// TIA Portal project "Control and SCADA Codes" (V20)
// Source code materials for the Control and SCADA Systems course.

(* hardware
DEVICE "S7-1500/ET200MP station_1"  S7-1500 station
   slot 0: "Rail_0"  Rack  6ES7 590-1***0-0AA0
   slot 1: "Control"  CPU 1511-1 PN  6ES7 511-1AL03-0AB0  V4.0
      slot 3: "CPU display_1"  6ES7591-1AA00-0AA0
      slot 32768: "PROFINET interface_1"  X1
         slot 32769: "Port_1"  X1 P1
         slot 32770: "Port_2"  X1 P2
      slot 34817: "Virtual CP interface port_1"  Virtual CP interface port  Virtual CP interface port FW V4.0
DEVICE "SCADA"  SIMATIC PC station
   slot 0: "SIMATIC PC station"  Rail  SIMATIC PC-Station  V1.0
      slot 125: "Stationmanager"  Station_Manager  V6.0.4
   slot 1: "HMI_RT_1"  WinCC Unified PC RT  6AV2 155-xxxxx-xxxx  20.0.0.0
DEVICE "S7-1500/ET200MP station_2"  S7-1500 station
   slot 0: "Rail_0"  Rack  6ES7 590-1***0-0AA0
   slot 1: "State Diagram Controller"  CPU 1511-1 PN  6ES7 511-1AL03-0AB0  V4.0
      slot 3: "CPU display_1"  6ES7591-1AA00-0AA0
      slot 32768: "PROFINET interface_1"  X1
         slot 32769: "Port_1"  X1 P1
         slot 32770: "Port_2"  X1 P2
      slot 34817: "Virtual CP interface port_1"  Virtual CP interface port  Virtual CP interface port FW V4.0
DEVICE "State Diagram SCADA"  SIMATIC PC station
   slot 0: "SIMATIC PC station"  Rail  SIMATIC PC-Station  V1.0
      slot 125: "Stationmanager"  Station_Manager  V6.0.4
   slot 1: "HMI_RT_2"  WinCC Unified PC RT  6AV2 155-xxxxx-xxxx  20.0.0.0
DEVICE "S7-1500/ET200MP station_3"  S7-1500 station
   slot 0: "Rail_0"  Rack  6ES7 590-1***0-0AA0
   slot 1: "OOP Controller"  CPU 1511-1 PN  6ES7 511-1AL03-0AB0  V4.0
      slot 3: "CPU display_1"  6ES7591-1AA00-0AA0
      slot 32768: "PROFINET interface_1"  X1
         slot 32769: "Port_1"  X1 P1
         slot 32770: "Port_2"  X1 P2
      slot 34817: "Virtual CP interface port_1"  Virtual CP interface port  Virtual CP interface port FW V4.0
DEVICE "OOP SCADA"  SIMATIC PC station
   slot 0: "SIMATIC PC station"  Rail  SIMATIC PC-Station  V1.0
      slot 125: "Stationmanager"  Station_Manager  V6.0.4
   slot 1: "HMI_RT_3"  WinCC Unified PC RT  6AV2 155-xxxxx-xxxx  20.0.0.0
DEVICE "S7-1500/ET200MP station_4"  S7-1500 station
   slot 0: "Rail_0"  Rack  6ES7 590-1***0-0AA0
   slot 1: "Contiuous Controller"  CPU 1511-1 PN  6ES7 511-1AL03-0AB0  V4.0
      slot 3: "CPU display_1"  6ES7591-1AA00-0AA0
      slot 32768: "PROFINET interface_1"  X1
         slot 32769: "Port_1"  X1 P1
         slot 32770: "Port_2"  X1 P2
      slot 34817: "Virtual CP interface port_1"  Virtual CP interface port  Virtual CP interface port FW V4.0
DEVICE "Continuous Ctrl SCADA"  SIMATIC PC station
   slot 0: "SIMATIC PC station"  Rail  SIMATIC PC-Station  V1.0
      slot 125: "Stationmanager"  Station_Manager  V6.0.4
   slot 1: "HMI_RT_4"  WinCC Unified PC RT  6AV2 155-xxxxx-xxxx  20.0.0.0
DEVICE "PC-System_1"  SIMATIC PC station
   slot 0: "SIMATIC PC station"  Rail  SIMATIC PC-Station  V1.0
      slot 125: "Stationmanager"  Station_Manager  V6.0.4
   slot 1: "Energy Management"  WinCC Unified PC RT  6AV2 155-xxxxx-xxxx  20.0.0.0
*)

// ===== PLC "Control"  CPU 1511-1 PN =====

VAR_GLOBAL   // PLC tag table "01.MotorCtrl"
   "Start" AT %M0.0 : Bool;
   "Stop" AT %M0.1 : Bool;
   "Motor" AT %M0.2 : Bool;
   "Clock_Byte" AT %MB100 : Byte;
   "Clock_10Hz" AT %M100.0 : Bool;
   "Clock_5Hz" AT %M100.1 : Bool;
   "Clock_2.5Hz" AT %M100.2 : Bool;
   "Clock_2Hz" AT %M100.3 : Bool;
   "Clock_1.25Hz" AT %M100.4 : Bool;
   "Clock_1Hz" AT %M100.5 : Bool;
   "Clock_0.625Hz" AT %M100.6 : Bool;
   "Clock_0.5Hz" AT %M100.7 : Bool;
END_VAR

VAR_GLOBAL   // PLC tag table "02.ThreeSwitchesCtrlPump"
   "K1" AT %M0.3 : Bool;
   "K2" AT %M0.4 : Bool;
   "K3" AT %M0.5 : Bool;
   "Pump" AT %M0.6 : Bool;
END_VAR

VAR_GLOBAL CONSTANT   // PLC tag table "02.ThreeSwitchesCtrlPump"
   "None(1)" : Pip := 65535;
   "Automatic update(1)" : Pip := 0;
   "PIP 1(1)" : Pip := 1;
   "PIP 2(1)" : Pip := 2;
   "PIP 3(1)" : Pip := 3;
   "PIP 4(1)" : Pip := 4;
   "PIP 5(1)" : Pip := 5;
   "PIP 6(1)" : Pip := 6;
   "PIP 7(1)" : Pip := 7;
   "PIP 8(1)" : Pip := 8;
   "PIP 9(1)" : Pip := 9;
   "PIP 10(1)" : Pip := 10;
   "PIP 11(1)" : Pip := 11;
   "PIP 12(1)" : Pip := 12;
   "PIP 13(1)" : Pip := 13;
   "PIP 14(1)" : Pip := 14;
   "PIP 15(1)" : Pip := 15;
   "PIP 16(1)" : Pip := 16;
   "PIP 17(1)" : Pip := 17;
   "PIP 18(1)" : Pip := 18;
   "PIP 19(1)" : Pip := 19;
   "PIP 20(1)" : Pip := 20;
   "PIP 21(1)" : Pip := 21;
   "PIP 22(1)" : Pip := 22;
   "PIP 23(1)" : Pip := 23;
   "PIP 24(1)" : Pip := 24;
   "PIP 25(1)" : Pip := 25;
   "PIP 26(1)" : Pip := 26;
   "PIP 27(1)" : Pip := 27;
   "PIP 28(1)" : Pip := 28;
   "PIP 29(1)" : Pip := 29;
   "PIP 30(1)" : Pip := 30;
   "PIP 31(1)" : Pip := 31;
   "PIP OB Servo(1)" : Pip := 32768;
   "Local~MC(1)" : Hw_SubModule := 51;
   "Local~Common(1)" : Hw_SubModule := 50;
   "Local~Device(1)" : Hw_Device := 32;
   "Local~Configuration(1)" : Hw_SubModule := 33;
   "Local~Display(1)" : Hw_SubModule := 54;
   "Local~Exec(1)" : Hw_SubModule := 52;
   "Local(1)" : Hw_SubModule := 49;
   "Local~PROFINET_interface_1(1)" : Hw_Interface := 64;
   "Local~PROFINET_interface_1~Port_1(1)" : Hw_Interface := 65;
   "Local~PROFINET_interface_1~Port_2(1)" : Hw_Interface := 66;
   "Local~Virtual_communication_interface(1)" : Hw_Interface := 135;
   "Local~License_Manager(1)" : Hw_SubModule := 42;
   "OB_01. MotorCtrl_LD(1)" : OB_PCYCLE := 1;
   "OB_02. MotorCtrl_FBD(1)" : OB_PCYCLE := 124;
   "OB_03. MotorCtrl_ST(1)" : OB_PCYCLE := 123;
   "OB_01_TheeSwitchesCtrlPump_1(1)" : OB_PCYCLE := 125;
END_VAR

VAR_GLOBAL   // PLC tag table "03.SBO"
   "Select" AT %M0.7 : Bool;
   "Confirm" AT %M1.0 : Bool;
   "CB" AT %M1.1 : Bool;
END_VAR

VAR_GLOBAL CONSTANT   // PLC tag table "03.SBO"
   "None(2)" : Pip := 65535;
   "Automatic update(2)" : Pip := 0;
   "PIP 1(2)" : Pip := 1;
   "PIP 2(2)" : Pip := 2;
   "PIP 3(2)" : Pip := 3;
   "PIP 4(2)" : Pip := 4;
   "PIP 5(2)" : Pip := 5;
   "PIP 6(2)" : Pip := 6;
   "PIP 7(2)" : Pip := 7;
   "PIP 8(2)" : Pip := 8;
   "PIP 9(2)" : Pip := 9;
   "PIP 10(2)" : Pip := 10;
   "PIP 11(2)" : Pip := 11;
   "PIP 12(2)" : Pip := 12;
   "PIP 13(2)" : Pip := 13;
   "PIP 14(2)" : Pip := 14;
   "PIP 15(2)" : Pip := 15;
   "PIP 16(2)" : Pip := 16;
   "PIP 17(2)" : Pip := 17;
   "PIP 18(2)" : Pip := 18;
   "PIP 19(2)" : Pip := 19;
   "PIP 20(2)" : Pip := 20;
   "PIP 21(2)" : Pip := 21;
   "PIP 22(2)" : Pip := 22;
   "PIP 23(2)" : Pip := 23;
   "PIP 24(2)" : Pip := 24;
   "PIP 25(2)" : Pip := 25;
   "PIP 26(2)" : Pip := 26;
   "PIP 27(2)" : Pip := 27;
   "PIP 28(2)" : Pip := 28;
   "PIP 29(2)" : Pip := 29;
   "PIP 30(2)" : Pip := 30;
   "PIP 31(2)" : Pip := 31;
   "PIP OB Servo(2)" : Pip := 32768;
   "Local~MC(2)" : Hw_SubModule := 51;
   "Local~Common(2)" : Hw_SubModule := 50;
   "Local~Device(2)" : Hw_Device := 32;
   "Local~Configuration(2)" : Hw_SubModule := 33;
   "Local~Display(2)" : Hw_SubModule := 54;
   "Local~Exec(2)" : Hw_SubModule := 52;
   "Local(2)" : Hw_SubModule := 49;
   "Local~PROFINET_interface_1(2)" : Hw_Interface := 64;
   "Local~PROFINET_interface_1~Port_1(2)" : Hw_Interface := 65;
   "Local~PROFINET_interface_1~Port_2(2)" : Hw_Interface := 66;
   "Local~Virtual_communication_interface(2)" : Hw_Interface := 135;
   "Local~License_Manager(2)" : Hw_SubModule := 42;
   "OB_01.MotorCtrl_LD(1)" : OB_PCYCLE := 1;
   "OB_02.MotorCtrl_FBD(1)" : OB_PCYCLE := 124;
   "OB_03.MotorCtrl_ST(1)" : OB_PCYCLE := 123;
   "OB_01_TheeSwitchesCtrlPump_1(2)" : OB_PCYCLE := 125;
   "OB_02_TheeSwitchesCtrlPump_2(1)" : OB_PCYCLE := 126;
   "OB_02.SBO_ST(1)" : OB_PCYCLE := 123;
   "OB_01.SBO_LD(1)" : OB_PCYCLE := 1;
END_VAR

VAR_GLOBAL   // PLC tag table "04.SafetyButton"
   "Progress" AT %MD2 : Time;
   "Press" AT %M1.2 : Bool;
   "LargeMotor" AT %M1.4 : Bool;
   "EStop" AT %M1.3 : Bool;
END_VAR

VAR_GLOBAL CONSTANT   // PLC tag table "04.SafetyButton"
   "None(3)" : Pip := 65535;
   "Automatic update(3)" : Pip := 0;
   "PIP 1(3)" : Pip := 1;
   "PIP 2(3)" : Pip := 2;
   "PIP 3(3)" : Pip := 3;
   "PIP 4(3)" : Pip := 4;
   "PIP 5(3)" : Pip := 5;
   "PIP 6(3)" : Pip := 6;
   "PIP 7(3)" : Pip := 7;
   "PIP 8(3)" : Pip := 8;
   "PIP 9(3)" : Pip := 9;
   "PIP 10(3)" : Pip := 10;
   "PIP 11(3)" : Pip := 11;
   "PIP 12(3)" : Pip := 12;
   "PIP 13(3)" : Pip := 13;
   "PIP 14(3)" : Pip := 14;
   "PIP 15(3)" : Pip := 15;
   "PIP 16(3)" : Pip := 16;
   "PIP 17(3)" : Pip := 17;
   "PIP 18(3)" : Pip := 18;
   "PIP 19(3)" : Pip := 19;
   "PIP 20(3)" : Pip := 20;
   "PIP 21(3)" : Pip := 21;
   "PIP 22(3)" : Pip := 22;
   "PIP 23(3)" : Pip := 23;
   "PIP 24(3)" : Pip := 24;
   "PIP 25(3)" : Pip := 25;
   "PIP 26(3)" : Pip := 26;
   "PIP 27(3)" : Pip := 27;
   "PIP 28(3)" : Pip := 28;
   "PIP 29(3)" : Pip := 29;
   "PIP 30(3)" : Pip := 30;
   "PIP 31(3)" : Pip := 31;
   "PIP OB Servo(3)" : Pip := 32768;
   "Local~MC(3)" : Hw_SubModule := 51;
   "Local~Common(3)" : Hw_SubModule := 50;
   "Local~Device(3)" : Hw_Device := 32;
   "Local~Configuration(3)" : Hw_SubModule := 33;
   "Local~Display(3)" : Hw_SubModule := 54;
   "Local~Exec(3)" : Hw_SubModule := 52;
   "Local(3)" : Hw_SubModule := 49;
   "Local~PROFINET_interface_1(3)" : Hw_Interface := 64;
   "Local~PROFINET_interface_1~Port_1(3)" : Hw_Interface := 65;
   "Local~PROFINET_interface_1~Port_2(3)" : Hw_Interface := 66;
   "Local~Virtual_communication_interface(3)" : Hw_Interface := 135;
   "Local~License_Manager(3)" : Hw_SubModule := 42;
   "OB_01.MotorCtrl_LD(2)" : OB_PCYCLE := 1;
   "OB_02.MotorCtrl_FBD(2)" : OB_PCYCLE := 124;
   "OB_03.MotorCtrl_ST(2)" : OB_PCYCLE := 123;
   "OB_01_TheeSwitchesCtrlPump_1(3)" : OB_PCYCLE := 125;
   "OB_02_TheeSwitchesCtrlPump_2(2)" : OB_PCYCLE := 126;
   "OB_02.SBO_ST(2)" : OB_PCYCLE := 123;
   "OB_01.SBO_LD(2)" : OB_PCYCLE := 1;
END_VAR

VAR_GLOBAL   // PLC tag table "05.CompressorService"
   "On" AT %M6.0 : Bool;
   "Off" AT %M6.1 : Bool;
   "Compressor" AT %M6.2 : Bool;
   "RunTime" AT %MD8 : Time;
   "AccTime" AT %MD12 : Time;
   "CycleCount" AT %MW16 : Int;
END_VAR

VAR_GLOBAL CONSTANT   // PLC tag table "05.CompressorService"
   "None(4)" : Pip := 65535;
   "Automatic update(4)" : Pip := 0;
   "PIP 1(4)" : Pip := 1;
   "PIP 2(4)" : Pip := 2;
   "PIP 3(4)" : Pip := 3;
   "PIP 4(4)" : Pip := 4;
   "PIP 5(4)" : Pip := 5;
   "PIP 6(4)" : Pip := 6;
   "PIP 7(4)" : Pip := 7;
   "PIP 8(4)" : Pip := 8;
   "PIP 9(4)" : Pip := 9;
   "PIP 10(4)" : Pip := 10;
   "PIP 11(4)" : Pip := 11;
   "PIP 12(4)" : Pip := 12;
   "PIP 13(4)" : Pip := 13;
   "PIP 14(4)" : Pip := 14;
   "PIP 15(4)" : Pip := 15;
   "PIP 16(4)" : Pip := 16;
   "PIP 17(4)" : Pip := 17;
   "PIP 18(4)" : Pip := 18;
   "PIP 19(4)" : Pip := 19;
   "PIP 20(4)" : Pip := 20;
   "PIP 21(4)" : Pip := 21;
   "PIP 22(4)" : Pip := 22;
   "PIP 23(4)" : Pip := 23;
   "PIP 24(4)" : Pip := 24;
   "PIP 25(4)" : Pip := 25;
   "PIP 26(4)" : Pip := 26;
   "PIP 27(4)" : Pip := 27;
   "PIP 28(4)" : Pip := 28;
   "PIP 29(4)" : Pip := 29;
   "PIP 30(4)" : Pip := 30;
   "PIP 31(4)" : Pip := 31;
   "PIP OB Servo(4)" : Pip := 32768;
   "Local~MC(4)" : Hw_SubModule := 51;
   "Local~Common(4)" : Hw_SubModule := 50;
   "Local~Device(4)" : Hw_Device := 32;
   "Local~Configuration(4)" : Hw_SubModule := 33;
   "Local~Display(4)" : Hw_SubModule := 54;
   "Local~Exec(4)" : Hw_SubModule := 52;
   "Local(4)" : Hw_SubModule := 49;
   "Local~PROFINET_interface_1(4)" : Hw_Interface := 64;
   "Local~PROFINET_interface_1~Port_1(4)" : Hw_Interface := 65;
   "Local~PROFINET_interface_1~Port_2(4)" : Hw_Interface := 66;
   "Local~Virtual_communication_interface(4)" : Hw_Interface := 135;
   "Local~License_Manager(4)" : Hw_SubModule := 42;
   "OB_01.MotorCtrl_LD(3)" : OB_PCYCLE := 1;
   "OB_02.MotorCtrl_FBD(3)" : OB_PCYCLE := 124;
   "OB_03.MotorCtrl_ST(3)" : OB_PCYCLE := 123;
   "OB_01_TheeSwitchesCtrlPump_1(4)" : OB_PCYCLE := 125;
   "OB_02_TheeSwitchesCtrlPump_2(3)" : OB_PCYCLE := 126;
   "OB_02.SBO_ST(3)" : OB_PCYCLE := 123;
   "OB_01.SBO_LD(3)" : OB_PCYCLE := 1;
END_VAR

VAR_GLOBAL   // PLC tag table "06.MotionSimulation"
   "OnCmd" AT %M18.0 : Bool;
   "OffCmd" AT %M18.1 : Bool;
   "Agitator" AT %M18.2 : Bool;
   "Rotor" AT %M22.0 : Bool;
   "Speed" AT %MD28 : Real;
   "Angle" AT %MD32 : Real;
   "Speed_SP" AT %MD24 : Real;
   "Position" AT %MW20 : Int;
END_VAR

VAR_GLOBAL CONSTANT   // PLC tag table "06.MotionSimulation"
   "None(5)" : Pip := 65535;
   "Automatic update(5)" : Pip := 0;
   "PIP 1(5)" : Pip := 1;
   "PIP 2(5)" : Pip := 2;
   "PIP 3(5)" : Pip := 3;
   "PIP 4(5)" : Pip := 4;
   "PIP 5(5)" : Pip := 5;
   "PIP 6(5)" : Pip := 6;
   "PIP 7(5)" : Pip := 7;
   "PIP 8(5)" : Pip := 8;
   "PIP 9(5)" : Pip := 9;
   "PIP 10(5)" : Pip := 10;
   "PIP 11(5)" : Pip := 11;
   "PIP 12(5)" : Pip := 12;
   "PIP 13(5)" : Pip := 13;
   "PIP 14(5)" : Pip := 14;
   "PIP 15(5)" : Pip := 15;
   "PIP 16(5)" : Pip := 16;
   "PIP 17(5)" : Pip := 17;
   "PIP 18(5)" : Pip := 18;
   "PIP 19(5)" : Pip := 19;
   "PIP 20(5)" : Pip := 20;
   "PIP 21(5)" : Pip := 21;
   "PIP 22(5)" : Pip := 22;
   "PIP 23(5)" : Pip := 23;
   "PIP 24(5)" : Pip := 24;
   "PIP 25(5)" : Pip := 25;
   "PIP 26(5)" : Pip := 26;
   "PIP 27(5)" : Pip := 27;
   "PIP 28(5)" : Pip := 28;
   "PIP 29(5)" : Pip := 29;
   "PIP 30(5)" : Pip := 30;
   "PIP 31(5)" : Pip := 31;
   "PIP OB Servo(5)" : Pip := 32768;
   "Local~MC(5)" : Hw_SubModule := 51;
   "Local~Common(5)" : Hw_SubModule := 50;
   "Local~Device(5)" : Hw_Device := 32;
   "Local~Configuration(5)" : Hw_SubModule := 33;
   "Local~Display(5)" : Hw_SubModule := 54;
   "Local~Exec(5)" : Hw_SubModule := 52;
   "Local(5)" : Hw_SubModule := 49;
   "Local~PROFINET_interface_1(5)" : Hw_Interface := 64;
   "Local~PROFINET_interface_1~Port_1(5)" : Hw_Interface := 65;
   "Local~PROFINET_interface_1~Port_2(5)" : Hw_Interface := 66;
   "Local~Virtual_communication_interface(5)" : Hw_Interface := 135;
   "Local~License_Manager(5)" : Hw_SubModule := 42;
   "OB_01.MotorCtrl_LD(4)" : OB_PCYCLE := 1;
   "OB_02.MotorCtrl_FBD(4)" : OB_PCYCLE := 124;
   "OB_03.MotorCtrl_ST(4)" : OB_PCYCLE := 123;
   "OB_01_TheeSwitchesCtrlPump_1(5)" : OB_PCYCLE := 125;
   "OB_02_TheeSwitchesCtrlPump_2(4)" : OB_PCYCLE := 126;
   "OB_02.SBO_ST(4)" : OB_PCYCLE := 123;
   "OB_01.SBO_LD(4)" : OB_PCYCLE := 1;
END_VAR

VAR_GLOBAL   // PLC tag table "07.2ndDiffEquationSim"
   "omega" AT %MD36 : Real;   // Tốc độ hiện tại (rad/s)
   "J" AT %MD48 : Real;   // Moment quán tính (kg.m^2)
   "B" AT %MD52 : Real;   // Hệ số ma sát nhớt (Nm.s/rad)
   "Kt" AT %MD56 : Real;   // Hệ số mô-men quay (Nm/A)
   "Ts" AT %MD60 : Real;   // Chu kỳ lấy mẫu (s)
   "i_in" AT %MD64 : Real;   // Dòng điện đầu vào (A)
   "alpha" AT %MD40 : Real;   // Gia tốc góc (rad/s^2)
   "theta" AT %MD44 : Real;   // vị trí góc
   "RunCmd" AT %M68.0 : Bool;
   "StopCmd" AT %M68.1 : Bool;
   "MotorStatus" AT %M68.2 : Bool;
   "MotorSpeed" AT %MD70 : Real;
   "MotorAngle" AT %MD74 : Real;
END_VAR

VAR_GLOBAL CONSTANT   // PLC tag table "07.2ndDiffEquationSim"
   "None(6)" : Pip := 65535;
   "Automatic update(6)" : Pip := 0;
   "PIP 1(6)" : Pip := 1;
   "PIP 2(6)" : Pip := 2;
   "PIP 3(6)" : Pip := 3;
   "PIP 4(6)" : Pip := 4;
   "PIP 5(6)" : Pip := 5;
   "PIP 6(6)" : Pip := 6;
   "PIP 7(6)" : Pip := 7;
   "PIP 8(6)" : Pip := 8;
   "PIP 9(6)" : Pip := 9;
   "PIP 10(6)" : Pip := 10;
   "PIP 11(6)" : Pip := 11;
   "PIP 12(6)" : Pip := 12;
   "PIP 13(6)" : Pip := 13;
   "PIP 14(6)" : Pip := 14;
   "PIP 15(6)" : Pip := 15;
   "PIP 16(6)" : Pip := 16;
   "PIP 17(6)" : Pip := 17;
   "PIP 18(6)" : Pip := 18;
   "PIP 19(6)" : Pip := 19;
   "PIP 20(6)" : Pip := 20;
   "PIP 21(6)" : Pip := 21;
   "PIP 22(6)" : Pip := 22;
   "PIP 23(6)" : Pip := 23;
   "PIP 24(6)" : Pip := 24;
   "PIP 25(6)" : Pip := 25;
   "PIP 26(6)" : Pip := 26;
   "PIP 27(6)" : Pip := 27;
   "PIP 28(6)" : Pip := 28;
   "PIP 29(6)" : Pip := 29;
   "PIP 30(6)" : Pip := 30;
   "PIP 31(6)" : Pip := 31;
   "PIP OB Servo(6)" : Pip := 32768;
   "Local~MC(6)" : Hw_SubModule := 51;
   "Local~Common(6)" : Hw_SubModule := 50;
   "Local~Device(6)" : Hw_Device := 32;
   "Local~Configuration(6)" : Hw_SubModule := 33;
   "Local~Display(6)" : Hw_SubModule := 54;
   "Local~Exec(6)" : Hw_SubModule := 52;
   "Local(6)" : Hw_SubModule := 49;
   "Local~PROFINET_interface_1(6)" : Hw_Interface := 64;
   "Local~PROFINET_interface_1~Port_1(6)" : Hw_Interface := 65;
   "Local~PROFINET_interface_1~Port_2(6)" : Hw_Interface := 66;
   "Local~Virtual_communication_interface(6)" : Hw_Interface := 135;
   "Local~License_Manager(6)" : Hw_SubModule := 42;
   "OB_01.MotorCtrl_LD(5)" : OB_PCYCLE := 1;
   "OB_02.MotorCtrl_FBD(5)" : OB_PCYCLE := 124;
   "OB_03.MotorCtrl_ST(5)" : OB_PCYCLE := 123;
   "OB_01_TheeSwitchesCtrlPump_1(6)" : OB_PCYCLE := 125;
   "OB_02_TheeSwitchesCtrlPump_2(5)" : OB_PCYCLE := 126;
   "OB_02.SBO_ST(5)" : OB_PCYCLE := 123;
   "OB_01.SBO_LD(5)" : OB_PCYCLE := 1;
END_VAR

// folder: System blocks/Program resources

DATA_BLOCK "SafetyDelay"   // DB1
{ S7_Optimized_Access := 'TRUE' }
AUTHOR : Simatic
FAMILY : IEC
NAME : IEC_TMR
VERSION : 1.0
// stored: InstanceOfName IEC_TIMER
"IEC_TIMER"
BEGIN
END_DATA_BLOCK

DATA_BLOCK "RunTimer"   // DB2
{ S7_Optimized_Access := 'TRUE' }
AUTHOR : Simatic
FAMILY : IEC
NAME : IEC_TMR
VERSION : 1.0
// stored: InstanceOfName IEC_TIMER
"IEC_TIMER"
BEGIN
END_DATA_BLOCK

DATA_BLOCK "AccTimer"   // DB3
{ S7_Optimized_Access := 'TRUE' }
AUTHOR : Simatic
FAMILY : IEC
NAME : IEC_TMR
VERSION : 1.0
// stored: InstanceOfName IEC_TIMER
"IEC_TIMER"
BEGIN
END_DATA_BLOCK

DATA_BLOCK "CycleCounter"   // DB4
{ S7_Optimized_Access := 'TRUE' }
AUTHOR : Simatic
FAMILY : IEC
NAME : CNTR
VERSION : 1.0
// stored: InstanceOfName IEC_COUNTER
"IEC_COUNTER"
BEGIN
END_DATA_BLOCK

DATA_BLOCK "PositionCounter"   // DB5
{ S7_Optimized_Access := 'TRUE' }
AUTHOR : Simatic
FAMILY : IEC
NAME : CNTR
VERSION : 1.0
// stored: InstanceOfName IEC_COUNTER
"IEC_COUNTER"
BEGIN
END_DATA_BLOCK

// folder: 01.Motor Ctrl

ORGANIZATION_BLOCK "01.MotorCtrl_LD"   // OB1, LAD, ProgramCycle
TITLE = "Main Program Sweep (Cycle)"
{ S7_Optimized_Access := 'TRUE' }
VERSION : 0.1
   VAR_INPUT
      Initial_Call : Bool;   // Initial call of this OB
      Remanence : Bool;   // =True, if remanent data are available
   END_VAR
BEGIN

REGION Network 1
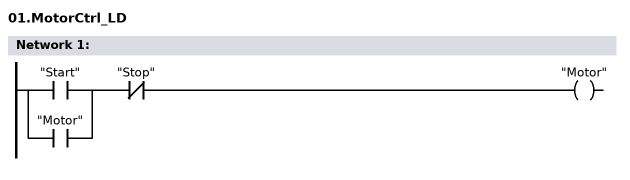
   RUNG wire#powerrail
      Contact( "Start" )
      wire#w1
      I_Contact( "Stop" )
      Coil( "Motor" )
   END_RUNG
   RUNG wire#powerrail
      Contact( "Motor" )
   END_RUNG wire#w1
   // the same network as SCL:
   "Motor" := ("Start" OR "Motor") AND NOT "Stop";
END_REGION
END_ORGANIZATION_BLOCK

ORGANIZATION_BLOCK "03.MotorCtrl_ST"   // OB123, SCL, ProgramCycle
TITLE = "Main Program Sweep (Cycle)"
{ S7_Optimized_Access := 'TRUE' }
VERSION : 0.1
   VAR_INPUT
      Initial_Call : Bool;   // Initial call of this OB
      Remanence : Bool;   // =True, if remanent data are available
   END_VAR
BEGIN
   "Motor" := ("Motor" OR "Start") AND NOT "Stop";
END_ORGANIZATION_BLOCK

ORGANIZATION_BLOCK "02.MotorCtrl_FBD"   // OB124, FBD, ProgramCycle
TITLE = "Main Program Sweep (Cycle)"
{ S7_Optimized_Access := 'TRUE' }
VERSION : 0.1
   VAR_INPUT
      Initial_Call : Bool;   // Initial call of this OB
      Remanence : Bool;   // =True, if remanent data are available
   END_VAR
BEGIN

REGION Network 1
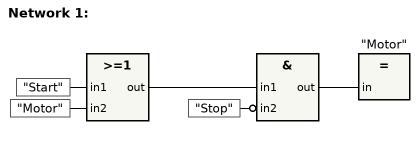
   "Motor" := ("Start" OR "Motor") AND NOT "Stop";
END_REGION
END_ORGANIZATION_BLOCK

// folder: 02.Three Switches Ctrl a Pump

ORGANIZATION_BLOCK "01_TheeSwitchesCtrlPump_1"   // OB125, SCL, ProgramCycle
TITLE = "Main Program Sweep (Cycle)"
{ S7_Optimized_Access := 'TRUE' }
VERSION : 0.1
   VAR_INPUT
      Initial_Call : Bool;   // Initial call of this OB
      Remanence : Bool;   // =True, if remanent data are available
   END_VAR
BEGIN
   (* Logic điều khiển bơm theo các tổ hợp của ba công tắc *)
   "Pump" := (NOT "K1" AND NOT "K2" AND "K3")
   OR (NOT "K1" AND "K2" AND NOT "K3")
   OR ("K1" AND NOT "K2" AND NOT "K3")
   OR ("K1" AND "K2" AND "K3");
END_ORGANIZATION_BLOCK

ORGANIZATION_BLOCK "02_TheeSwitchesCtrlPump_2"   // OB126, SCL, ProgramCycle
TITLE = "Main Program Sweep (Cycle)"
{ S7_Optimized_Access := 'TRUE' }
VERSION : 0.1
   VAR_INPUT
      Initial_Call : Bool;   // Initial call of this OB
      Remanence : Bool;   // =True, if remanent data are available
   END_VAR
BEGIN
   (* Logic điều khiển bơm sử dụng XOR *)
   "Pump" := "K1" XOR "K2" XOR "K3";
END_ORGANIZATION_BLOCK

// folder: 03.SBO

ORGANIZATION_BLOCK "01.SBO_LD"   // OB127, LAD, ProgramCycle
TITLE = "Main Program Sweep (Cycle)"
{ S7_Optimized_Access := 'TRUE' }
VERSION : 0.1
   VAR_INPUT
      Initial_Call : Bool;   // Initial call of this OB
      Remanence : Bool;   // =True, if remanent data are available
   END_VAR
BEGIN

REGION Network 1
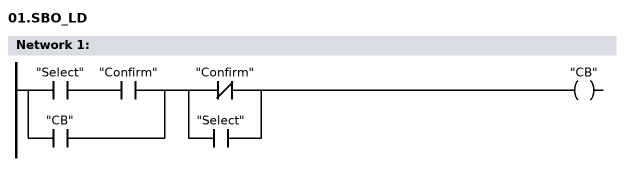
   RUNG wire#powerrail
      Contact( "Select" )
      Contact( "Confirm" )
      wire#w1
      I_Contact( "Confirm" )
      wire#w2
      Coil( "CB" )
   END_RUNG
   RUNG wire#powerrail
      Contact( "CB" )
   END_RUNG wire#w1
   RUNG wire#w1
      Contact( "Select" )
   END_RUNG wire#w2
   // the same network as SCL:
   "CB" := (("Select" AND "Confirm") OR "CB") AND (NOT "Confirm" OR "Select");
END_REGION
END_ORGANIZATION_BLOCK

ORGANIZATION_BLOCK "02.SBO_ST"   // OB128, SCL, ProgramCycle
TITLE = "Main Program Sweep (Cycle)"
{ S7_Optimized_Access := 'TRUE' }
VERSION : 0.1
   VAR_INPUT
      Initial_Call : Bool;   // Initial call of this OB
      Remanence : Bool;   // =True, if remanent data are available
   END_VAR
BEGIN
   "Motor" := ("Motor" OR "Start") AND NOT "Stop";
END_ORGANIZATION_BLOCK

// folder: 04.Safety Button

ORGANIZATION_BLOCK "01.SafetyButton_LD"   // OB129, LAD, ProgramCycle
TITLE = "Main Program Sweep (Cycle)"
{ S7_Optimized_Access := 'TRUE' }
VERSION : 0.1
   VAR_INPUT
      Initial_Call : Bool;   // Initial call of this OB
      Remanence : Bool;   // =True, if remanent data are available
   END_VAR
BEGIN

REGION Network 1
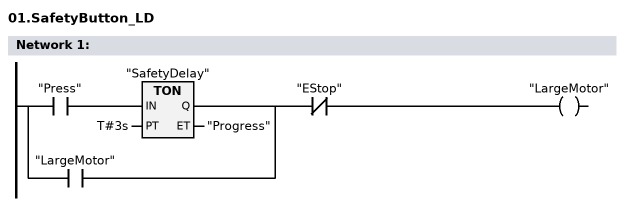
   "SafetyDelay".TON(IN := "Press", PT := T#3s, ET => "Progress");
   "LargeMotor" := ("SafetyDelay".Q OR "LargeMotor") AND NOT "EStop";
END_REGION
END_ORGANIZATION_BLOCK

ORGANIZATION_BLOCK "03.SafetyButton_ST"   // OB130, SCL, ProgramCycle
TITLE = "Main Program Sweep (Cycle)"
{ S7_Optimized_Access := 'TRUE' }
VERSION : 0.1
   VAR_INPUT
      Initial_Call : Bool;   // Initial call of this OB
      Remanence : Bool;   // =True, if remanent data are available
   END_VAR
BEGIN
   "SafetyDelay".TON(IN := "Press",
                     PT:=T#3s);
   "LargeMotor" := ("LargeMotor" OR "SafetyDelay".Q) AND NOT "EStop";
END_ORGANIZATION_BLOCK

ORGANIZATION_BLOCK "02.SafetyButton_FBD"   // OB131, FBD, ProgramCycle
TITLE = "Main Program Sweep (Cycle)"
{ S7_Optimized_Access := 'TRUE' }
VERSION : 0.1
   VAR_INPUT
      Initial_Call : Bool;   // Initial call of this OB
      Remanence : Bool;   // =True, if remanent data are available
   END_VAR
BEGIN

REGION Network 1
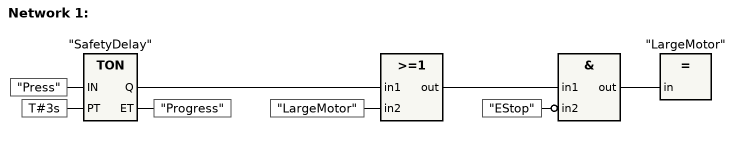
   "SafetyDelay".TON(IN := "Press", PT := T#3s, ET => "Progress");
   "LargeMotor" := ("SafetyDelay".Q OR "LargeMotor") AND NOT "EStop";
END_REGION
END_ORGANIZATION_BLOCK

// folder: 05.Compressor Service

ORGANIZATION_BLOCK "02.CompressorService_ST"   // OB132, SCL, ProgramCycle
TITLE = "Main Program Sweep (Cycle)"
{ S7_Optimized_Access := 'TRUE' }
VERSION : 0.1
   VAR_INPUT
      Initial_Call : Bool;   // Initial call of this OB
      Remanence : Bool;   // =True, if remanent data are available
   END_VAR
BEGIN
   "Compressor" := ("Compressor" OR "On") AND NOT "Off";
   "RunTimer".TON(IN:="Compressor",
                  PT:=T#24D,
                  ET => "RunTime");

   "AccTimer".TONR(IN := "Compressor",
                  PT := T#24D,
                  ET => "AccTime");

   "CycleCounter".CTU(CU := "Compressor",
                  PV := 32767,
                  CV => "CycleCount");
END_ORGANIZATION_BLOCK

ORGANIZATION_BLOCK "01.CompressorService_FBD"   // OB133, FBD, ProgramCycle
TITLE = "Main Program Sweep (Cycle)"
{ S7_Optimized_Access := 'TRUE' }
VERSION : 0.1
   VAR_INPUT
      Initial_Call : Bool;   // Initial call of this OB
      Remanence : Bool;   // =True, if remanent data are available
   END_VAR
BEGIN

REGION Network 1
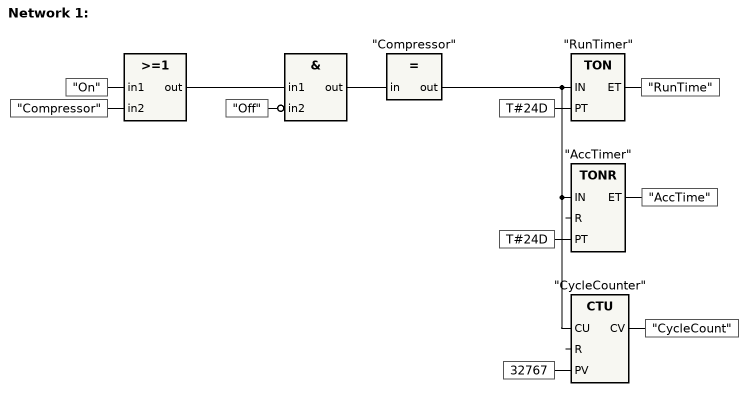
   "Compressor" := ("On" OR "Compressor") AND NOT "Off";
   "RunTimer".TON(IN := "Compressor", PT := T#24D, ET => "RunTime");
   "AccTimer".TONR(IN := "Compressor", PT := T#24D, ET => "AccTime");
   "CycleCounter".CTU(CU := "Compressor", PV := 32767, CV => "CycleCount");
END_REGION
END_ORGANIZATION_BLOCK

// folder: 06.Motion Simulation

ORGANIZATION_BLOCK "01.MotionSimulation"   // OB134, FBD, ProgramCycle
TITLE = "Main Program Sweep (Cycle)"
{ S7_Optimized_Access := 'TRUE' }
VERSION : 0.1
   VAR_INPUT
      Initial_Call : Bool;   // Initial call of this OB
      Remanence : Bool;   // =True, if remanent data are available
   END_VAR
BEGIN

REGION Network 1
   // Control and Agitator postion simulation
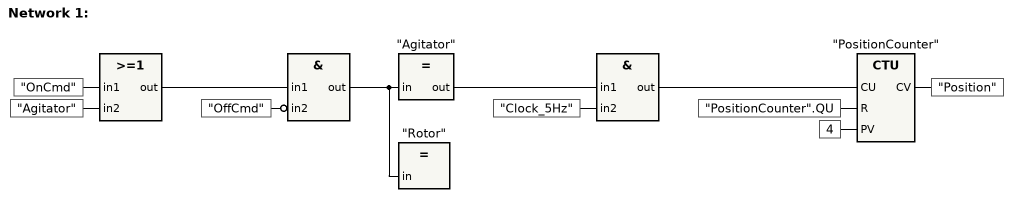
   "Agitator" := ("OnCmd" OR "Agitator") AND NOT "OffCmd";
   "PositionCounter".CTU(CU := "Agitator" AND "Clock_5Hz", R := "PositionCounter".QU, PV := 4, CV => "Position");
   "Rotor" := "Agitator";
END_REGION

REGION Network 2 (SCL)
   // Speed and Angle Simulation
   "R_TRIG_10Hz"(CLK:="Clock_10Hz");

   (* Cập nhật tốc độ Speed mỗi 100 ms *)
   IF "R_TRIG_10Hz".Q THEN
       IF "Rotor" THEN
           IF "Speed" < "Speed_SP" THEN
               "Speed" := "Speed" + 10;
               IF "Speed" > "Speed_SP" THEN
                   "Speed" := "Speed_SP";
               END_IF;
           ELSE
               "Speed" := "Speed" - 20;
               IF "Speed" < "Speed_SP" THEN
                   "Speed" := "Speed_SP";
               END_IF;
           END_IF;
       ELSE
           "Speed" := "Speed" - 25;
           IF "Speed" < 0 THEN
               "Speed" := 0;
           END_IF;
       END_IF;

       (* Cập nhật góc quay *)
       "Angle" := "Angle" + (25 * "Speed") / 1000;
       IF "Angle" >= 360 THEN
           "Angle" := 0;
       END_IF;
   END_IF;
END_REGION
END_ORGANIZATION_BLOCK

// ===== PLC "State Diagram Controller"  CPU 1511-1 PN =====

VAR_GLOBAL   // PLC tag table "01.Tank"
   "Start" AT %M0.0 : Bool;
   "Stop" AT %M0.1 : Bool;
   "Lo" AT %M0.2 : Bool;
   "Hi" AT %M0.3 : Bool;
   "P_1" AT %M0.4 : Bool;
   "P_2" AT %M0.5 : Bool;
   "P_3" AT %M0.6 : Bool;
   "T01" AT %M0.7 : Bool;
   "T12" AT %M1.0 : Bool;
   "T24" AT %M1.2 : Bool;
   "T34" AT %M1.3 : Bool;
   "T42" AT %M1.4 : Bool;
   "T21" AT %M1.5 : Bool;
   "T31" AT %M1.6 : Bool;
   "T41" AT %M1.7 : Bool;
   "S1" AT %M2.0 : Bool;
   "S2" AT %M2.1 : Bool;
   "S3" AT %M2.2 : Bool;
   "S4" AT %M2.3 : Bool;
   "L" AT %MW4 : Int;
   "T23" AT %M1.1 : Bool;
END_VAR

VAR_GLOBAL   // PLC tag table "02.BatchControl"
   "StartBatch" AT %M10.0 : Bool;
   "StopBatch" AT %M10.1 : Bool;
   "High" AT %M10.2 : Bool;
   "Low" AT %M10.3 : Bool;
   "Mixer" AT %M10.4 : Bool;
   "Pump_A" AT %M10.5 : Bool;
   "Pump_B" AT %M10.6 : Bool;
   "Pump_P" AT %M10.7 : Bool;
   "T_01" AT %M11.0 : Bool;
   "T_12" AT %M11.1 : Bool;
   "T_23" AT %M11.2 : Bool;
   "T_34" AT %M11.3 : Bool;
   "T_45" AT %M11.4 : Bool;
   "T_56" AT %M11.5 : Bool;
   "T_61" AT %M11.6 : Bool;
   "T_62" AT %M11.7 : Bool;
   "T_21" AT %M12.0 : Bool;
   "T_31" AT %M12.1 : Bool;
   "T_41" AT %M12.2 : Bool;
   "T_51" AT %M12.3 : Bool;
   "S_1" AT %M12.4 : Bool;
   "S_2" AT %M12.5 : Bool;
   "S_3" AT %M12.6 : Bool;
   "S_4" AT %M12.7 : Bool;
   "S_5" AT %M13.0 : Bool;
   "S_6" AT %M13.1 : Bool;
   "BatchActive" AT %M13.2 : Bool;
   "Va" AT %MD14 : Real;
   "Vb" AT %MD18 : Real;
   "Va_SP" AT %MD22 : Real;
   "Vb_SP" AT %MD26 : Real;
   "ProductCnt" AT %MW30 : Int;
   "ProductCnt_SP" AT %MW32 : Int;
   "Level" AT %MW34 : Int;
END_VAR

VAR_GLOBAL CONSTANT   // PLC tag table "02.BatchControl"
   "None(1)" : Pip := 65535;
   "Automatic update(1)" : Pip := 0;
   "PIP 1(1)" : Pip := 1;
   "PIP 2(1)" : Pip := 2;
   "PIP 3(1)" : Pip := 3;
   "PIP 4(1)" : Pip := 4;
   "PIP 5(1)" : Pip := 5;
   "PIP 6(1)" : Pip := 6;
   "PIP 7(1)" : Pip := 7;
   "PIP 8(1)" : Pip := 8;
   "PIP 9(1)" : Pip := 9;
   "PIP 10(1)" : Pip := 10;
   "PIP 11(1)" : Pip := 11;
   "PIP 12(1)" : Pip := 12;
   "PIP 13(1)" : Pip := 13;
   "PIP 14(1)" : Pip := 14;
   "PIP 15(1)" : Pip := 15;
   "PIP 16(1)" : Pip := 16;
   "PIP 17(1)" : Pip := 17;
   "PIP 18(1)" : Pip := 18;
   "PIP 19(1)" : Pip := 19;
   "PIP 20(1)" : Pip := 20;
   "PIP 21(1)" : Pip := 21;
   "PIP 22(1)" : Pip := 22;
   "PIP 23(1)" : Pip := 23;
   "PIP 24(1)" : Pip := 24;
   "PIP 25(1)" : Pip := 25;
   "PIP 26(1)" : Pip := 26;
   "PIP 27(1)" : Pip := 27;
   "PIP 28(1)" : Pip := 28;
   "PIP 29(1)" : Pip := 29;
   "PIP 30(1)" : Pip := 30;
   "PIP 31(1)" : Pip := 31;
   "PIP OB Servo(1)" : Pip := 32768;
   "Local~MC(1)" : Hw_SubModule := 51;
   "Local~Common(1)" : Hw_SubModule := 50;
   "Local~Device(1)" : Hw_Device := 32;
   "Local~Configuration(1)" : Hw_SubModule := 33;
   "Local~Display(1)" : Hw_SubModule := 54;
   "Local~Exec(1)" : Hw_SubModule := 52;
   "Local(1)" : Hw_SubModule := 49;
   "Local~PROFINET_interface_1(1)" : Hw_Interface := 64;
   "Local~PROFINET_interface_1~Port_1(1)" : Hw_Interface := 65;
   "Local~PROFINET_interface_1~Port_2(1)" : Hw_Interface := 66;
   "Local~Virtual_communication_interface(1)" : Hw_Interface := 135;
   "Local~License_Manager(1)" : Hw_SubModule := 42;
   "OB_01.PumpControl(1)" : OB_PCYCLE := 1;
   "OB_02.LevelSim(1)" : OB_PCYCLE := 123;
END_VAR

VAR_GLOBAL   // PLC tag table "@System"
   "Clock_Byte" AT %MB100 : Byte;
   "Clock_10Hz" AT %M100.0 : Bool;
   "Clock_5Hz" AT %M100.1 : Bool;
   "Clock_2.5Hz" AT %M100.2 : Bool;
   "Clock_2Hz" AT %M100.3 : Bool;
   "Clock_1.25Hz" AT %M100.4 : Bool;
   "Clock_1Hz" AT %M100.5 : Bool;
   "Clock_0.625Hz" AT %M100.6 : Bool;
   "Clock_0.5Hz" AT %M100.7 : Bool;
   "System_Byte" AT %MB101 : Byte;
   "FirstScan" AT %M101.0 : Bool;
   "DiagStatusUpdate" AT %M101.1 : Bool;
   "AlwaysTRUE" AT %M101.2 : Bool;
   "AlwaysFALSE" AT %M101.3 : Bool;
END_VAR

VAR_GLOBAL CONSTANT   // PLC tag table "@System"
   "None(2)" : Pip := 65535;
   "Automatic update(2)" : Pip := 0;
   "PIP 1(2)" : Pip := 1;
   "PIP 2(2)" : Pip := 2;
   "PIP 3(2)" : Pip := 3;
   "PIP 4(2)" : Pip := 4;
   "PIP 5(2)" : Pip := 5;
   "PIP 6(2)" : Pip := 6;
   "PIP 7(2)" : Pip := 7;
   "PIP 8(2)" : Pip := 8;
   "PIP 9(2)" : Pip := 9;
   "PIP 10(2)" : Pip := 10;
   "PIP 11(2)" : Pip := 11;
   "PIP 12(2)" : Pip := 12;
   "PIP 13(2)" : Pip := 13;
   "PIP 14(2)" : Pip := 14;
   "PIP 15(2)" : Pip := 15;
   "PIP 16(2)" : Pip := 16;
   "PIP 17(2)" : Pip := 17;
   "PIP 18(2)" : Pip := 18;
   "PIP 19(2)" : Pip := 19;
   "PIP 20(2)" : Pip := 20;
   "PIP 21(2)" : Pip := 21;
   "PIP 22(2)" : Pip := 22;
   "PIP 23(2)" : Pip := 23;
   "PIP 24(2)" : Pip := 24;
   "PIP 25(2)" : Pip := 25;
   "PIP 26(2)" : Pip := 26;
   "PIP 27(2)" : Pip := 27;
   "PIP 28(2)" : Pip := 28;
   "PIP 29(2)" : Pip := 29;
   "PIP 30(2)" : Pip := 30;
   "PIP 31(2)" : Pip := 31;
   "PIP OB Servo(2)" : Pip := 32768;
   "Local~MC(2)" : Hw_SubModule := 51;
   "Local~Common(2)" : Hw_SubModule := 50;
   "Local~Device(2)" : Hw_Device := 32;
   "Local~Configuration(2)" : Hw_SubModule := 33;
   "Local~Display(2)" : Hw_SubModule := 54;
   "Local~Exec(2)" : Hw_SubModule := 52;
   "Local(2)" : Hw_SubModule := 49;
   "Local~PROFINET_interface_1(2)" : Hw_Interface := 64;
   "Local~PROFINET_interface_1~Port_1(2)" : Hw_Interface := 65;
   "Local~PROFINET_interface_1~Port_2(2)" : Hw_Interface := 66;
   "Local~Virtual_communication_interface(2)" : Hw_Interface := 135;
   "Local~License_Manager(2)" : Hw_SubModule := 42;
   "OB_01.PumpControl(2)" : OB_PCYCLE := 1;
   "OB_02.LevelSim(2)" : OB_PCYCLE := 123;
   "OB_01.BatchControl(1)" : OB_PCYCLE := 124;
   "OB_02.TankSim(1)" : OB_PCYCLE := 125;
   "OB_03.ProductDetectSim(1)" : OB_PCYCLE := 126;
END_VAR

// folder: System blocks/Program resources

DATA_BLOCK "TON_5s"   // DB1
{ S7_Optimized_Access := 'TRUE' }
AUTHOR : Simatic
FAMILY : IEC
NAME : IEC_TMR
VERSION : 1.0
// stored: InstanceOfName IEC_TIMER
"IEC_TIMER"
BEGIN
END_DATA_BLOCK

DATA_BLOCK "TON_20s"   // DB2
{ S7_Optimized_Access := 'TRUE' }
AUTHOR : Simatic
FAMILY : IEC
NAME : IEC_TMR
VERSION : 1.0
// stored: InstanceOfName IEC_TIMER
"IEC_TIMER"
BEGIN
END_DATA_BLOCK

DATA_BLOCK "ProductCounter"   // DB4
{ S7_Optimized_Access := 'TRUE' }
AUTHOR : Simatic
FAMILY : IEC
NAME : CNTR
VERSION : 1.0
// stored: InstanceOfName IEC_COUNTER
"IEC_COUNTER"
BEGIN
END_DATA_BLOCK

DATA_BLOCK "TON_10s"   // DB8
{ S7_Optimized_Access := 'TRUE' }
AUTHOR : Simatic
FAMILY : IEC
NAME : IEC_TMR
VERSION : 1.0
// stored: InstanceOfName IEC_TIMER
"IEC_TIMER"
BEGIN
END_DATA_BLOCK

// folder: 01. Tank

ORGANIZATION_BLOCK "01.PumpControl"   // OB1, SCL, ProgramCycle
TITLE = "Main Program Sweep (Cycle)"
{ S7_Optimized_Access := 'TRUE' }
VERSION : 0.1
   VAR_INPUT
      Initial_Call : Bool;   // Initial call of this OB
      Remanence : Bool;   // =True, if remanent data are available
   END_VAR
BEGIN

   // Timer 10s (đang ở chế độ nạp 1 bơm)
   "TON_10s".TON(IN := "S2", PT := T#10S);

   // Phương trình TRANSITION
   "T01" := "FirstScan";
   "T12" := "S1" AND "Start";
   "T23" := "S2" AND "TON_10s".Q AND NOT "Hi";
   "T24" := "S2" AND "Hi";
   "T34" := "S3" AND "Hi";
   "T42" := "S4" AND "Lo";
   "T21" := "S2" AND "Stop";
   "T31" := "S3" AND "Stop";
   "T41" := "S4" AND "Stop";

   // Phương trình TRẠNG THÁI
   "S1" := ("S1" OR "T01" OR "T21" OR "T31" OR "T41") AND NOT "T12";
   "S2" := ("S2" OR "T12" OR "T42") AND NOT "T23" AND NOT "T24" AND NOT "T21";
   "S3" := ("S3" OR "T23") AND NOT "T34" AND NOT "T31";
   "S4" := ("S4" OR "T24" OR "T34") AND NOT "T42" AND NOT "T41";

   // Phương trình OUTPUT
   "P_1" := "S2" OR "S3";
   "P_2" := "S3";
   "P_3" := "S4";
END_ORGANIZATION_BLOCK

ORGANIZATION_BLOCK "02.LevelSim"   // OB123, SCL, ProgramCycle
TITLE = "Main Program Sweep (Cycle)"
{ S7_Optimized_Access := 'TRUE' }
VERSION : 0.1
   VAR_INPUT
      Initial_Call : Bool;   // Initial call of this OB
      Remanence : Bool;   // =True, if remanent data are available
   END_VAR
   VAR_TEMP
      dL : Int;
   END_VAR
BEGIN
   "R_TRIG_1Hz"(CLK := "Clock_1Hz");
   IF "R_TRIG_1Hz".Q THEN
       #dL := 5 * BOOL_TO_INT("P_1") + 5 * BOOL_TO_INT("P_2") - 10 * BOOL_TO_INT("P_3");
       "L" := "L" + #dL;
       IF "L" > 100 THEN
           "L" := 100;
       ELSIF "L" < 0 THEN
           "L" := 0;
       END_IF;
       "Hi" := ("L" > 98);
       "Lo" := ("L" < 2);
   END_IF;
END_ORGANIZATION_BLOCK

// folder: 02. Batch Control

ORGANIZATION_BLOCK "01.BatchControl"   // OB124, SCL, ProgramCycle
TITLE = "Main Program Sweep (Cycle)"
{ S7_Optimized_Access := 'TRUE' }
VERSION : 0.1
   VAR_INPUT
      Initial_Call : Bool;   // Initial call of this OB
      Remanence : Bool;   // =True, if remanent data are available
   END_VAR
BEGIN
   // Timer 5s (trong trạng thái S_2)
   "TON_5s".TON(IN := "S_6", PT := T#5S);

   // Timer 20s (trong trạng thái S_4 - Mixer)
   "TON_20s".TON(IN := "S_4", PT := T#20S);

   // Phương trình TRANSITION
   "T_01" := "FirstScan";
   "T_12" := "S_1" AND "StartBatch";
   "T_23" := "S_2" AND ("Va" >= "Va_SP");
   "T_34" := "S_3" AND ("Vb" >= "Vb_SP");
   "T_45" := "S_4" AND "TON_20s".Q;
   "T_56" := "S_5" AND "Low";
   "T_61" := "S_6" AND ("StopBatch" OR ("ProductCnt" >= "ProductCnt_SP"));
   "T_62" := "S_6" AND (NOT "StopBatch") AND ("ProductCnt" < "ProductCnt_SP") AND "TON_5s".Q;

   "T_21" := "S_2" AND ("StopBatch" AND "High");
   "T_31" := "S_3" AND ("StopBatch" AND "High");
   "T_41" := "S_4" AND "StopBatch";
   "T_51" := "S_5" AND "StopBatch";

   // Phương trình TRẠNG THÁI
   "S_1" := ("S_1" OR "T_01" OR "T_21" OR "T_31" OR "T_41" OR "T_51" OR "T_61") AND NOT "T_12";
   "S_2" := ("S_2" OR "T_12" OR "T_62") AND NOT "T_23" AND NOT "T_21";
   "S_3" := ("S_3" OR "T_23") AND NOT "T_34" AND NOT "T_31";
   "S_4" := ("S_4" OR "T_34") AND NOT "T_45" AND NOT "T_41";
   "S_5" := ("S_5" OR "T_45") AND NOT "T_56" AND NOT "T_51";
   "S_6" := ("S_6" OR "T_56") AND NOT "T_61" AND NOT "T_62";

   // Phương trình OUTPUT
   "Pump_A" := "S_2";
   "Pump_B" := "S_3";
   "Mixer" := "S_4";
   "Pump_P" := "S_5";
END_ORGANIZATION_BLOCK

ORGANIZATION_BLOCK "02.TankSim"   // OB125, SCL, ProgramCycle
TITLE = "Main Program Sweep (Cycle)"
{ S7_Optimized_Access := 'TRUE' }
VERSION : 0.1
   VAR_INPUT
      Initial_Call : Bool;   // Initial call of this OB
      Remanence : Bool;   // =True, if remanent data are available
   END_VAR
   VAR_TEMP
      dVa_in : Real;
      dVb_in : Real;
      dV_out : Real;
      fa : Real;
      fb : Real;
      Vt : Real;
   END_VAR
   VAR CONSTANT
      Qa : Real := 1.75;
      Qb : Real := 1.25;
      Qp : Real := 3.15;
      C : Real := 100.0;
   END_VAR
BEGIN
   // Trigger theo xung 1Hz
   "R_TRIG_2Hz"(CLK := "Clock_2Hz");

   IF "R_TRIG_2Hz".Q THEN

       // Tính dòng vào/ra
       #dVa_in := #Qa * BOOL_TO_INT("Pump_A");
       #dVb_in := #Qb * BOOL_TO_INT("Pump_B");
       #dV_out := #Qp * BOOL_TO_INT("Pump_P");

       // Tính phần trăm thành phần
       IF ("Va" + "Vb") > 0.0 THEN
           #fa := "Va" / ("Va" + "Vb");
           #fb := "Vb" / ("Va" + "Vb");
       ELSE
           #fa := 0.0;
           #fb := 0.0;
       END_IF;

       // Cập nhật thể tích A và B
       "Va" := "Va" + #dVa_in - #fa * #dV_out;
       "Vb" := "Vb" + #dVb_in - #fb * #dV_out;

       // Giới hạn thể tích
       IF "Va" < 0.0 THEN
           "Va" := 0.0;
       END_IF;
       IF "Vb" < 0.0 THEN
           "Vb" := 0.0;
       END_IF;
       IF "Va" > #C THEN
           "Va" := #C;
       END_IF;
       IF "Vb" > #C THEN
           "Vb" := #C;
       END_IF;

       // Tổng thể tích và mức
       #Vt := "Va" + "Vb";
       "Level" := 100.0 * #Vt / #C;

       // Ngưỡng mức
       "High" := ("Level" > 98.0);
       "Low" := ("Level" < 2.0);
   END_IF;
END_ORGANIZATION_BLOCK

ORGANIZATION_BLOCK "03.ProductDetectSim"   // OB126, SCL, ProgramCycle
TITLE = "Main Program Sweep (Cycle)"
{ S7_Optimized_Access := 'TRUE' }
VERSION : 0.1
   VAR_INPUT
      Initial_Call : Bool;   // Initial call of this OB
      Remanence : Bool;   // =True, if remanent data are available
   END_VAR
BEGIN
   "BatchActive" := ("BatchActive" OR "StartBatch") AND NOT "StopBatch";

   "R_TRIG_Low"(CLK := "Low");

   "ProductCounter".CTU(CU:="BatchActive" AND "R_TRIG_Low".Q,
                        PV:="ProductCnt_SP", R := "S_1", CV => "ProductCnt");
END_ORGANIZATION_BLOCK

// ===== PLC "OOP Controller"  CPU 1511-1 PN =====

VAR_GLOBAL   // PLC tag table "@System Tags"
   "Clock_Byte" AT %MB100 : Byte;
   "Clock_10Hz" AT %M100.0 : Bool;
   "Clock_5Hz" AT %M100.1 : Bool;
   "Clock_2.5Hz" AT %M100.2 : Bool;
   "Clock_2Hz" AT %M100.3 : Bool;
   "Clock_1.25Hz" AT %M100.4 : Bool;
   "Clock_1Hz" AT %M100.5 : Bool;
   "Clock_0.625Hz" AT %M100.6 : Bool;
   "Clock_0.5Hz" AT %M100.7 : Bool;
   "System_Byte" AT %MB101 : Byte;
   "FirstScan" AT %M101.0 : Bool;
   "DiagStatusUpdate" AT %M101.1 : Bool;
   "AlwaysTRUE" AT %M101.2 : Bool;
   "AlwaysFALSE" AT %M101.3 : Bool;
END_VAR

VAR_GLOBAL   // PLC tag table "01.Tank"
   "Start" AT %M0.0 : Bool;
   "Stop" AT %M0.1 : Bool;
   "Lo" AT %M0.2 : Bool;
   "Hi" AT %M0.3 : Bool;
   "P_1" AT %M0.4 : Bool;
   "P_2" AT %M0.5 : Bool;
   "P_3" AT %M0.6 : Bool;
   "T01" AT %M0.7 : Bool;
   "T12" AT %M1.0 : Bool;
   "T24" AT %M1.2 : Bool;
   "T34" AT %M1.3 : Bool;
   "T42" AT %M1.4 : Bool;
   "T21" AT %M1.5 : Bool;
   "T31" AT %M1.6 : Bool;
   "T41" AT %M1.7 : Bool;
   "S1" AT %M2.0 : Bool;
   "S2" AT %M2.1 : Bool;
   "S3" AT %M2.2 : Bool;
   "S4" AT %M2.3 : Bool;
   "L" AT %MW4 : Int;
   "T23" AT %M1.1 : Bool;
END_VAR

VAR_GLOBAL CONSTANT   // PLC tag table "01.Tank"
   "None(1)" : Pip := 65535;
   "Automatic update(1)" : Pip := 0;
   "PIP 1(1)" : Pip := 1;
   "PIP 2(1)" : Pip := 2;
   "PIP 3(1)" : Pip := 3;
   "PIP 4(1)" : Pip := 4;
   "PIP 5(1)" : Pip := 5;
   "PIP 6(1)" : Pip := 6;
   "PIP 7(1)" : Pip := 7;
   "PIP 8(1)" : Pip := 8;
   "PIP 9(1)" : Pip := 9;
   "PIP 10(1)" : Pip := 10;
   "PIP 11(1)" : Pip := 11;
   "PIP 12(1)" : Pip := 12;
   "PIP 13(1)" : Pip := 13;
   "PIP 14(1)" : Pip := 14;
   "PIP 15(1)" : Pip := 15;
   "PIP 16(1)" : Pip := 16;
   "PIP 17(1)" : Pip := 17;
   "PIP 18(1)" : Pip := 18;
   "PIP 19(1)" : Pip := 19;
   "PIP 20(1)" : Pip := 20;
   "PIP 21(1)" : Pip := 21;
   "PIP 22(1)" : Pip := 22;
   "PIP 23(1)" : Pip := 23;
   "PIP 24(1)" : Pip := 24;
   "PIP 25(1)" : Pip := 25;
   "PIP 26(1)" : Pip := 26;
   "PIP 27(1)" : Pip := 27;
   "PIP 28(1)" : Pip := 28;
   "PIP 29(1)" : Pip := 29;
   "PIP 30(1)" : Pip := 30;
   "PIP 31(1)" : Pip := 31;
   "PIP OB Servo(1)" : Pip := 32768;
   "Local~MC(1)" : Hw_SubModule := 51;
   "Local~Common(1)" : Hw_SubModule := 50;
   "Local~Device(1)" : Hw_Device := 32;
   "Local~Configuration(1)" : Hw_SubModule := 33;
   "Local~Display(1)" : Hw_SubModule := 54;
   "Local~Exec(1)" : Hw_SubModule := 52;
   "Local(1)" : Hw_SubModule := 49;
   "Local~PROFINET_interface_1(1)" : Hw_Interface := 64;
   "Local~PROFINET_interface_1~Port_1(1)" : Hw_Interface := 65;
   "Local~PROFINET_interface_1~Port_2(1)" : Hw_Interface := 66;
   "Local~Virtual_communication_interface(1)" : Hw_Interface := 135;
   "Local~License_Manager(1)" : Hw_SubModule := 42;
   "OB_01.PumpControl" : OB_PCYCLE := 1;
   "OB_02.LevelSim" : OB_PCYCLE := 123;
   "OB_01.BatchControl" : OB_PCYCLE := 124;
   "OB_02.TankSim" : OB_PCYCLE := 125;
   "OB_03.ProductDetectSim" : OB_PCYCLE := 126;
END_VAR

// folder: 01. Flate2Object

DATA_BLOCK "SimpleMotor_1"   // DB1
{ S7_Optimized_Access := 'FALSE' }
VERSION : 0.1
// stored: InstanceOfName SimpleMotor
"SimpleMotor"
BEGIN
END_DATA_BLOCK

DATA_BLOCK "SimpleMotor_2"   // DB2
{ S7_Optimized_Access := 'FALSE' }
VERSION : 0.1
// stored: InstanceOfName SimpleMotor
"SimpleMotor"
BEGIN
END_DATA_BLOCK

DATA_BLOCK "SimpleMotor_3"   // DB3
{ S7_Optimized_Access := 'FALSE' }
VERSION : 0.1
// stored: InstanceOfName SimpleMotor
"SimpleMotor"
BEGIN
END_DATA_BLOCK

// folder: 02. Full OOP

DATA_BLOCK "Motor_1"   // DB4
{ S7_Optimized_Access := 'FALSE' }
VERSION : 0.1
// stored: InstanceOfName Motor
"Motor"
BEGIN
END_DATA_BLOCK

DATA_BLOCK "Motor_2"   // DB5
{ S7_Optimized_Access := 'FALSE' }
VERSION : 0.1
// stored: InstanceOfName Motor
"Motor"
BEGIN
END_DATA_BLOCK

DATA_BLOCK "Motor_3"   // DB6
{ S7_Optimized_Access := 'FALSE' }
VERSION : 0.1
// stored: InstanceOfName Motor
"Motor"
BEGIN
END_DATA_BLOCK

// folder: System blocks/Program resources

DATA_BLOCK "TON_10s"   // DB7
{ S7_Optimized_Access := 'TRUE' }
AUTHOR : Simatic
FAMILY : IEC
NAME : IEC_TMR
VERSION : 1.0
// stored: InstanceOfName IEC_TIMER
"IEC_TIMER"
BEGIN
END_DATA_BLOCK

// folder: 01. Flate2Object

FUNCTION_BLOCK "SimpleMotor"   // FB1, SCL
{ S7_Optimized_Access := 'FALSE' }
VERSION : 0.1
   VAR_INPUT
      Start : Bool;
      Stop : Bool;
   END_VAR
   VAR_OUTPUT
      Cmd : Bool;
   END_VAR
   VAR_IN_OUT
      Test : Bool;
   END_VAR
BEGIN
   #Cmd := (#Cmd OR #Start) AND NOT #Stop;
END_FUNCTION_BLOCK

ORGANIZATION_BLOCK "SimpleMotorInstances"   // OB1, FBD, ProgramCycle
TITLE = "Main Program Sweep (Cycle)"
{ S7_Optimized_Access := 'TRUE' }
VERSION : 0.1
   VAR_INPUT
      Initial_Call : Bool;   // Initial call of this OB
      Remanence : Bool;   // =True, if remanent data are available
   END_VAR
BEGIN

REGION Network 1
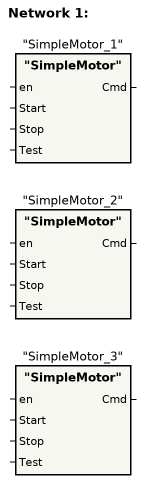
   "SimpleMotor_1"();   // "SimpleMotor"
   "SimpleMotor_2"();   // "SimpleMotor"
   "SimpleMotor_3"();   // "SimpleMotor"
END_REGION
END_ORGANIZATION_BLOCK

// folder: 02. Full OOP

FUNCTION_BLOCK "Motor"   // FB2, SCL
{ S7_Optimized_Access := 'FALSE' }
VERSION : 0.1
   VAR_INPUT
      Mode : Int;   // 0 - MAN, 1 - AUTO
      Start : Bool;
      Stop : Bool;
      Start_Aut : Bool;
      Stop_Aut : Bool;
      RunFb : Bool;
      Reset : Bool;
      Speed_SP : Real;
   END_VAR
   VAR_OUTPUT
      Cmd : Bool;
      Fault : Bool;
      Runtime : Time;
      Speed : Real;
      Angle : Real;
   END_VAR
   VAR
      Runtimer : TON_TIME;
      CmdDelay : TON_TIME;
      R_TRIG_10Hz : R_TRIG;
   END_VAR
BEGIN
   IF #Mode = 0 THEN
       #Cmd := (#Start OR #Cmd) AND NOT #Stop AND NOT #Fault;
   END_IF;

   IF #Mode = 1 THEN
       #Cmd := (#Start_Aut OR #Cmd) AND NOT #Stop_Aut AND NOT #Fault;
   END_IF;

   #CmdDelay(IN:=#Cmd,
             PT:=T#10S);

   IF #CmdDelay.Q AND NOT #RunFb THEN
       #Fault := TRUE;
   END_IF;

   IF #Reset THEN
       #Fault := FALSE;
   END_IF;

   #Runtimer(IN:=#RunFb,
             PT:=T#24D,
             ET=>#Runtime);

   #R_TRIG_10Hz(CLK:="Clock_10Hz");

   (* Cập nhật tốc độ Speed mỗi 100 ms *)
   IF #R_TRIG_10Hz.Q THEN
       IF #RunFb THEN
           IF #Speed<#Speed_SP THEN
               #Speed:=#Speed + 10;
               IF #Speed>#Speed_SP THEN
                   #Speed:=#Speed_SP;
               END_IF;
           ELSE
               #Speed:=#Speed - 20;
               IF #Speed<#Speed_SP THEN
                   #Speed:=#Speed_SP;
               END_IF;
           END_IF;
       ELSE
           #Speed:=#Speed - 25;
           IF #Speed < 0 THEN
               #Speed := 0;
           END_IF;
       END_IF;

       (* Cập nhật góc quay *)
       #Angle:=#Angle+ (25 *#Speed) / 1000;
       IF #Angle >= 360 THEN
           #Angle := 0;
       END_IF;
   END_IF;
END_FUNCTION_BLOCK

ORGANIZATION_BLOCK "PnID"   // OB123, FBD, ProgramCycle
TITLE = "Main Program Sweep (Cycle)"
{ S7_Optimized_Access := 'TRUE' }
VERSION : 0.1
   VAR_INPUT
      Initial_Call : Bool;   // Initial call of this OB
      Remanence : Bool;   // =True, if remanent data are available
   END_VAR
BEGIN

REGION Network 1
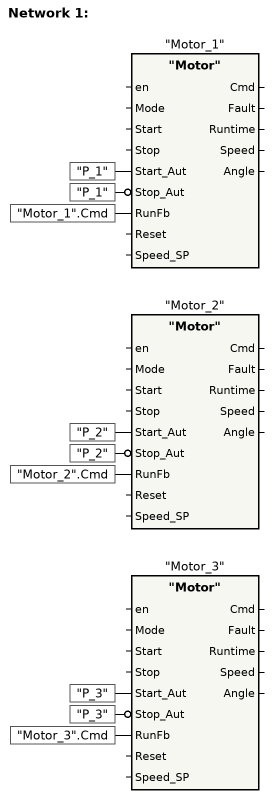
   "Motor_1"(Start_Aut := "P_1", Stop_Aut := NOT "P_1", RunFb := "Motor_1".Cmd);   // "Motor"
   "Motor_2"(Start_Aut := "P_2", Stop_Aut := NOT "P_2", RunFb := "Motor_2".Cmd);   // "Motor"
   "Motor_3"(Start_Aut := "P_3", Stop_Aut := NOT "P_3", RunFb := "Motor_3".Cmd);   // "Motor"
END_REGION
END_ORGANIZATION_BLOCK

// folder: 03. OOPxStateDiagram

ORGANIZATION_BLOCK "01.PumpControl"   // OB124, SCL, ProgramCycle
TITLE = "Main Program Sweep (Cycle)"
{ S7_Optimized_Access := 'TRUE' }
VERSION : 0.1
   VAR_INPUT
      Initial_Call : Bool;   // Initial call of this OB
      Remanence : Bool;   // =True, if remanent data are available
   END_VAR
BEGIN

   // Timer 10s (đang ở chế độ nạp 1 bơm)
   "TON_10s".TON(IN := "S2", PT := T#10S);

   // Phương trình TRANSITION
   "T01" := "FirstScan";
   "T12" := "S1" AND "Start";
   "T23" := "S2" AND "TON_10s".Q AND NOT "Hi";
   "T24" := "S2" AND "Hi";
   "T34" := "S3" AND "Hi";
   "T42" := "S4" AND "Lo";
   "T21" := "S2" AND "Stop";
   "T31" := "S3" AND "Stop";
   "T41" := "S4" AND "Stop";

   // Phương trình TRẠNG THÁI
   "S1" := ("S1" OR "T01" OR "T21" OR "T31" OR "T41") AND NOT "T12";
   "S2" := ("S2" OR "T12" OR "T42") AND NOT "T23" AND NOT "T24" AND NOT "T21";
   "S3" := ("S3" OR "T23") AND NOT "T34" AND NOT "T31";
   "S4" := ("S4" OR "T24" OR "T34") AND NOT "T42" AND NOT "T41";

   // Phương trình OUTPUT
   "P_1" := "S2" OR "S3";
   "P_2" := "S3";
   "P_3" := "S4";
END_ORGANIZATION_BLOCK

ORGANIZATION_BLOCK "02.LevelSim"   // OB125, SCL, ProgramCycle
TITLE = "Main Program Sweep (Cycle)"
{ S7_Optimized_Access := 'TRUE' }
VERSION : 0.1
   VAR_INPUT
      Initial_Call : Bool;   // Initial call of this OB
      Remanence : Bool;   // =True, if remanent data are available
   END_VAR
   VAR_TEMP
      dL : Int;
   END_VAR
BEGIN
   "R_TRIG_1Hz"(CLK := "Clock_1Hz");

   IF "R_TRIG_1Hz".Q THEN
       #dL := 5 * BOOL_TO_INT("Motor_1".RunFb) + 5 * BOOL_TO_INT("Motor_2".RunFb) - 10 * BOOL_TO_INT("Motor_3".RunFb);
       "L" := "L" + #dL;
       IF "L" > 100 THEN
           "L" := 100;
       ELSIF "L" < 0 THEN
           "L" := 0;
       END_IF;
       "Hi" := ("L" > 98);
       "Lo" := ("L" < 2);
   END_IF;
END_ORGANIZATION_BLOCK

// ===== PLC "Contiuous Controller"  CPU 1511-1 PN =====

VAR_GLOBAL   // PLC tag table "@System Tags"
   "Clock_Byte" AT %MB100 : Byte;
   "Clock_10Hz" AT %M100.0 : Bool;
   "Clock_5Hz" AT %M100.1 : Bool;
   "Clock_2.5Hz" AT %M100.2 : Bool;
   "Clock_2Hz" AT %M100.3 : Bool;
   "Clock_1.25Hz" AT %M100.4 : Bool;
   "Clock_1Hz" AT %M100.5 : Bool;
   "Clock_0.625Hz" AT %M100.6 : Bool;
   "Clock_0.5Hz" AT %M100.7 : Bool;
   "System_Byte" AT %MB101 : Byte;
   "FirstScan" AT %M101.0 : Bool;
   "DiagStatusUpdate" AT %M101.1 : Bool;
   "AlwaysTRUE" AT %M101.2 : Bool;
   "AlwaysFALSE" AT %M101.3 : Bool;
END_VAR

VAR_GLOBAL CONSTANT   // PLC tag table "01.Tank"
   "None(1)" : Pip := 65535;
   "Automatic update(1)" : Pip := 0;
   "PIP 1(1)" : Pip := 1;
   "PIP 2(1)" : Pip := 2;
   "PIP 3(1)" : Pip := 3;
   "PIP 4(1)" : Pip := 4;
   "PIP 5(1)" : Pip := 5;
   "PIP 6(1)" : Pip := 6;
   "PIP 7(1)" : Pip := 7;
   "PIP 8(1)" : Pip := 8;
   "PIP 9(1)" : Pip := 9;
   "PIP 10(1)" : Pip := 10;
   "PIP 11(1)" : Pip := 11;
   "PIP 12(1)" : Pip := 12;
   "PIP 13(1)" : Pip := 13;
   "PIP 14(1)" : Pip := 14;
   "PIP 15(1)" : Pip := 15;
   "PIP 16(1)" : Pip := 16;
   "PIP 17(1)" : Pip := 17;
   "PIP 18(1)" : Pip := 18;
   "PIP 19(1)" : Pip := 19;
   "PIP 20(1)" : Pip := 20;
   "PIP 21(1)" : Pip := 21;
   "PIP 22(1)" : Pip := 22;
   "PIP 23(1)" : Pip := 23;
   "PIP 24(1)" : Pip := 24;
   "PIP 25(1)" : Pip := 25;
   "PIP 26(1)" : Pip := 26;
   "PIP 27(1)" : Pip := 27;
   "PIP 28(1)" : Pip := 28;
   "PIP 29(1)" : Pip := 29;
   "PIP 30(1)" : Pip := 30;
   "PIP 31(1)" : Pip := 31;
   "PIP OB Servo(1)" : Pip := 32768;
   "Local~MC(1)" : Hw_SubModule := 51;
   "Local~Common(1)" : Hw_SubModule := 50;
   "Local~Device(1)" : Hw_Device := 32;
   "Local~Configuration(1)" : Hw_SubModule := 33;
   "Local~Display(1)" : Hw_SubModule := 54;
   "Local~Exec(1)" : Hw_SubModule := 52;
   "Local(1)" : Hw_SubModule := 49;
   "Local~PROFINET_interface_1(1)" : Hw_Interface := 64;
   "Local~PROFINET_interface_1~Port_1(1)" : Hw_Interface := 65;
   "Local~PROFINET_interface_1~Port_2(1)" : Hw_Interface := 66;
   "Local~Virtual_communication_interface(1)" : Hw_Interface := 135;
   "Local~License_Manager(1)" : Hw_SubModule := 42;
   "OB_01.PumpControl" : OB_PCYCLE := 1;
   "OB_02.LevelSim" : OB_PCYCLE := 123;
   "OB_01.BatchControl" : OB_PCYCLE := 124;
   "OB_02.TankSim" : OB_PCYCLE := 125;
   "OB_03.ProductDetectSim" : OB_PCYCLE := 126;
END_VAR

// folder: 01. Heater

DATA_BLOCK "ON_OFF_Ctrl_1"   // DB1
{ S7_Optimized_Access := 'TRUE' }
VERSION : 0.1
// stored: InstanceOfName ON_OFF_Ctrl
"ON_OFF_Ctrl"
BEGIN
END_DATA_BLOCK

DATA_BLOCK "HeaterSim_1"   // DB2
{ S7_Optimized_Access := 'FALSE' }
VERSION : 0.1
// stored: InstanceOfName HeaterSim
"HeaterSim"
BEGIN
END_DATA_BLOCK

// folder: 02. Motor

DATA_BLOCK "MotorSim_1"   // DB4
{ S7_Optimized_Access := 'FALSE' }
VERSION : 0.1
// stored: InstanceOfName MotorSim
"MotorSim"
BEGIN
END_DATA_BLOCK

DATA_BLOCK "DOL_Ctrl_1"   // DB5
{ S7_Optimized_Access := 'FALSE' }
VERSION : 0.1
// stored: InstanceOfName DOL_Ctrl
"DOL_Ctrl"
BEGIN
END_DATA_BLOCK

// folder: 03. PID

DATA_BLOCK "PID_100"   // DB6
{ S7_Optimized_Access := 'FALSE' }
VERSION : 0.1
// stored: InstanceOfName PID
"PID"
BEGIN
END_DATA_BLOCK

DATA_BLOCK "HeaterSim_100"   // DB7
{ S7_Optimized_Access := 'FALSE' }
VERSION : 0.1
// stored: InstanceOfName HeaterSim
"HeaterSim"
BEGIN
END_DATA_BLOCK

DATA_BLOCK "MotorSim_101"   // DB8
{ S7_Optimized_Access := 'FALSE' }
VERSION : 0.1
// stored: InstanceOfName MotorSim
"MotorSim"
BEGIN
END_DATA_BLOCK

DATA_BLOCK "DOL_101"   // DB9
{ S7_Optimized_Access := 'FALSE' }
VERSION : 0.1
// stored: InstanceOfName DOL_Ctrl
"DOL_Ctrl"
BEGIN
END_DATA_BLOCK

DATA_BLOCK "PID_101"   // DB10
{ S7_Optimized_Access := 'FALSE' }
VERSION : 0.1
// stored: InstanceOfName PID
"PID"
BEGIN
END_DATA_BLOCK

// folder: 01. Heater

FUNCTION_BLOCK "HeaterSim"   // FB1, SCL
{ S7_Optimized_Access := 'FALSE' }
VERSION : 0.1
   VAR_INPUT
      Enable : Bool;
      Tamb : Real := 25.0;
      HeaterOn : Bool;
      Tick : Bool;
   END_VAR
   VAR_OUTPUT
      T : Real := 25.0;
      Ready : Bool;
      Fault : Bool;
   END_VAR
   VAR
      T1 : Real := 25.0;
   END_VAR
   VAR_TEMP
      "a" : Real;
      "b" : Real;
      u : Real;
   END_VAR
   VAR CONSTANT
      Ts : Real := 0.1;
      Tau : Real := 60.0;
      K : Real := 120.0;
      Tmin : Real := 0.0;
      Tmax : Real := 300.0;
   END_VAR
BEGIN
   // FB sẵn sàng
   #Ready := TRUE;

   IF #Enable AND #Tick THEN

       // Chuyển tín hiệu DOL sang dạng số
       IF #HeaterOn THEN
           #u := 1.0;
       ELSE
           #u := 0.0;
       END_IF;

       // Hệ số rời rạc
       #a := #Ts / #Tau;
       #b := (#Ts / #Tau) * #K;

       // Cập nhật nhiệt độ
       #T := (1.0 - #a) * #T1 + #a * #Tamb + #b * #u;

       // Giới hạn nhiệt độ
       IF #T < #Tmin THEN
           #T := #Tmin;
       END_IF;
       IF #T > #Tmax THEN
           #T := #Tmax;
       END_IF;

       // Lưu trạng thái
       #T1 := #T;

       // Cảnh báo quá nhiệt (tùy chọn)
       #Fault := (#T >= (#Tmax - 1.0));

   END_IF;
END_FUNCTION_BLOCK

FUNCTION_BLOCK "ON_OFF_Ctrl"   // FB2, FBD
{ S7_Optimized_Access := 'TRUE' }
VERSION : 0.1
   VAR_INPUT
      Enable : Bool;
      T : Real;
      SP : Real := 80.0;
      Hys : Real := 2.0;
   END_VAR
   VAR_OUTPUT
      HeaterOn : Bool;
   END_VAR
BEGIN

REGION Network 1 (SCL)
   // Điều khiển DOL có hysteresis
   IF NOT #Enable THEN
       #HeaterOn := FALSE;
   ELSE
       // Điều kiện bật gia nhiệt
       IF (NOT #HeaterOn) AND (#T <= (#SP - #Hys)) THEN
           #HeaterOn := TRUE;
       END_IF;

       // Điều kiện tắt gia nhiệt
       IF #HeaterOn AND (#T >= (#SP + #Hys)) THEN
           #HeaterOn := FALSE;
       END_IF;
   END_IF;
END_REGION
END_FUNCTION_BLOCK

ORGANIZATION_BLOCK "ONOFFCtrl"   // OB1, SCL, ProgramCycle
TITLE = "Main Program Sweep (Cycle)"
{ S7_Optimized_Access := 'TRUE' }
VERSION : 0.1
   VAR_INPUT
      Initial_Call : Bool;   // Initial call of this OB
      Remanence : Bool;   // =True, if remanent data are available
   END_VAR
BEGIN
   "R_TRIG_10Hz"(CLK := "Clock_10Hz");

   "ON_OFF_Ctrl_1"(T        := "HeaterSim_1".T,
           Hys      := 2.0);

   "HeaterSim_1"(
              Enable := TRUE,
              HeaterOn := "ON_OFF_Ctrl_1".HeaterOn,
              Tick := "R_TRIG_10Hz".Q);
END_ORGANIZATION_BLOCK

// folder: 02. Motor

FUNCTION_BLOCK "MotorSim"   // FB3, SCL
{ S7_Optimized_Access := 'FALSE' }
VERSION : 0.1
   VAR_INPUT
      Enable : Bool;
      Run : Bool;
      i_in : Real;
      Tick : Bool;
   END_VAR
   VAR_OUTPUT
      Omega : Real;
      Theta : Real;
      Ready : Bool;
      Fault : Bool;
   END_VAR
   VAR
      omega_1 : Real;
      theta_1 : Real;
   END_VAR
   VAR_TEMP
      alpha : Real;
      i_eff : Real;
   END_VAR
   VAR CONSTANT
      Ts : Real := 0.1;
      J : Real := 0.25;
      "B" : Real := 0.3;
      Kt : Real := 0.628;
      omega_max : Real := 300.0;
   END_VAR
BEGIN
   // FB sẵn sàng
   #Ready := TRUE;

   IF #Enable AND #Tick THEN

       // Xác định dòng kích thích
       IF #Run THEN
           #i_eff := #i_in;
       ELSE
           #i_eff := 0.0;
       END_IF;

       // Gia tốc góc
       #alpha := (#Kt * #i_eff - #B * #omega_1) / #J;

       // Cập nhật vận tốc
       #Omega := #omega_1 + #Ts * #alpha;

       // Giới hạn tốc độ
       IF #Omega > #omega_max THEN
           #Omega := #omega_max;
       END_IF;
       IF #Omega < 0.0 THEN
           #Omega := 0.0;
       END_IF;

       // Cập nhật vị trí
       #Theta := #theta_1 + #Ts * #Omega;

       // Lưu trạng thái
       #omega_1 := #Omega;
       #theta_1 := #Theta;

       // Cảnh báo quá tốc
       #Fault := (#Omega >= #omega_max);

   END_IF;
END_FUNCTION_BLOCK

FUNCTION_BLOCK "DOL_Ctrl"   // FB4, FBD
{ S7_Optimized_Access := 'FALSE' }
VERSION : 0.1
   VAR_INPUT
      Enable : Bool;
      RunCmd : Bool;
      i_set : Real := 80.0;
   END_VAR
   VAR_OUTPUT
      Run : Bool;
      i_out : Real;
   END_VAR
BEGIN

REGION Network 1 (SCL)
   // Điều khiển DOL
   IF NOT #Enable THEN
       #Run := FALSE;
       #i_out := 0.0;
   ELSE
       IF #RunCmd THEN
           #Run := TRUE;
           #i_out := #i_set;
       ELSE
           #Run := FALSE;
           #i_out := 0.0;
       END_IF;
   END_IF;
END_REGION
END_FUNCTION_BLOCK

ORGANIZATION_BLOCK "DOLCtrl"   // OB123, SCL, ProgramCycle
TITLE = "Main Program Sweep (Cycle)"
{ S7_Optimized_Access := 'TRUE' }
VERSION : 0.1
   VAR_INPUT
      Initial_Call : Bool;   // Initial call of this OB
      Remanence : Bool;   // =True, if remanent data are available
   END_VAR
BEGIN
   "DOL_Ctrl_1"(
                Enable := "MotorSim_1".Ready
   );

   "MotorSim_1"(
                Enable := TRUE,
                Run := "DOL_Ctrl_1".Run,
                i_in := "DOL_Ctrl_1".i_out,
                Tick := "R_TRIG_10Hz".Q
   );
END_ORGANIZATION_BLOCK

// folder: 03. PID

FUNCTION_BLOCK "PID"   // FB5, SCL
{ S7_Optimized_Access := 'FALSE' }
VERSION : 0.1
   VAR_INPUT
      Enable : Bool;
      SP : Real;
      PV : Real;
      Tick : Bool;
      Kp : Real;
      Ki : Real;
      Kd : Real;
      u_min : Real;
      u_max : Real;
   END_VAR
   VAR_OUTPUT
      u : Real;
      Ready : Bool;
   END_VAR
   VAR
      e_1 : Real;
      "e" : Real;
      I : Real;
      P : Real;
      D : Real;
   END_VAR
   VAR_TEMP
      u_raw : Real;
   END_VAR
   VAR CONSTANT
      Ts : Real := 0.1;
   END_VAR
BEGIN
   #Ready := TRUE;

   IF #Enable AND #Tick THEN
       // Sai lệch
       #e := #SP - #PV;

       // P
       #P := #Kp * #e;

       // I
       #I := #I + #Ki * #Ts * #e;

       // D
       #D := #Kd * (#e - #e_1) / #Ts;

       // Tổng hợp
       #u_raw := #P + #I + #D;

       // Giới hạn ngõ ra
       #u := #u_raw;
       IF #u > #u_max THEN
           #u := #u_max;
       END_IF;
       IF #u < #u_min THEN
           #u := #u_min;
       END_IF;

       // Chống bão hòa tích phân
       IF #u <> #u_raw THEN
           #I := #I - #Ki * #Ts * #e;
       END_IF;

       // Lưu trạng thái
       #e_1 := #e;

   END_IF;
END_FUNCTION_BLOCK

ORGANIZATION_BLOCK "HeaterPIDCtrl"   // OB124, SCL, ProgramCycle
TITLE = "Main Program Sweep (Cycle)"
{ S7_Optimized_Access := 'TRUE' }
VERSION : 0.1
   VAR_INPUT
      Initial_Call : Bool;   // Initial call of this OB
      Remanence : Bool;   // =True, if remanent data are available
   END_VAR
   VAR_TEMP
      pid_out : Real;
      HeaterOn : Bool;
   END_VAR
BEGIN
   // Bộ điều khiển PID
   "PID_100"(
             PV := "HeaterSim_100".T,
             Tick := "R_TRIG_10Hz".Q,

             Kp := 2.0,
             Ki := 0.1,
             Kd := 0.0,

             u_min := -100.0,
             u_max := 100.0,
             u      => #pid_out
   );

   // Ánh xạ PID sang tín hiệu gia nhiệt
   IF #pid_out > 0.0 THEN
       #HeaterOn := TRUE;
   ELSE
       #HeaterOn := FALSE;
   END_IF;


   "HeaterSim_100"(
                 Enable := TRUE,
                 HeaterOn := #HeaterOn,
                 Tick := "R_TRIG_10Hz".Q);
END_ORGANIZATION_BLOCK

ORGANIZATION_BLOCK "MotorPIDCtrl"   // OB125, SCL, ProgramCycle
TITLE = "Main Program Sweep (Cycle)"
{ S7_Optimized_Access := 'TRUE' }
VERSION : 0.1
   VAR_INPUT
      Initial_Call : Bool;   // Initial call of this OB
      Remanence : Bool;   // =True, if remanent data are available
   END_VAR
BEGIN
   // Bộ điều khiển PID tốc độ
   "PID_101"(
             PV     := "MotorSim_101".Omega,
             Tick   := "R_TRIG_10Hz".Q,

             u_min  := 0.0,
             u_max  := 150.0
   );

   // Điều khiển chạy/dừng động cơ (DOL)
   "DOL_101"(
             Enable := "MotorSim_101".Ready);

   // Mô phỏng động cơ
   "MotorSim_101"(
                  Enable := TRUE,
                  Run    := "DOL_101".Run,
                  i_in   := "PID_101".u,
                  Tick   := "R_TRIG_10Hz".Q
   );
END_ORGANIZATION_BLOCK

(* ===== HMI "HMI_RT_1" =====
connection "Connection_1": ETHERNET, ILRT_S7_1500_OMS

HMI tags "01.MotorCtrl"
   "Start" : Bool AT %M0.0, T100ms
   "Stop" : Bool AT %M0.1, T100ms
   "Motor" : Bool AT %M0.2, T100ms

HMI tags "02.ThreeSwitchesCtrPump"
   "K2" : Bool AT %M0.4, T100ms
   "K3" : Bool AT %M0.5, T100ms
   "K1" : Bool AT %M0.3, T100ms
   "Pump" : Bool AT %M0.6, T100ms

HMI tags "03.SBO"
   "Confirm" : Bool AT %M1.0, T100ms
   "CB" : Bool AT %M1.1, T100ms
   "Select" : Bool AT %M0.7, T100ms

HMI tags "04.SafetyButton"
   "Progress" : Time AT %MD2, T100ms
   "LargeMotor" : Bool AT %M1.4, T100ms
   "EStop" : Bool AT %M1.3, T100ms
   "Press" : Bool AT %M1.2, T100ms

HMI tags "05.CompressorService"
   "RunTime" : DInt AT %MD8, T100ms
   "Off" : Bool AT %M6.1, T100ms
   "On" : Bool AT %M6.0, T100ms
   "Compressor" : Bool AT %M6.2, T100ms
   "AccTime" : DInt AT %MD12, T100ms
   "CycleCount" : Int AT %MW16, T100ms

HMI tags "06.MotionSimulation"
   "Speed_SP" : Real AT %MD24, T100ms
   "Position" : Int AT %MW20, T100ms
   "Rotor" : Bool AT %M22.0, T100ms
   "OffCmd" : Bool AT %M18.1, T100ms
   "OnCmd" : Bool AT %M18.0, T100ms
   "Agitator" : Bool AT %M18.2, T100ms
   "Speed" : Real AT %MD28, T100ms
   "Angle" : Real AT %MD32, T100ms

text list "SystemTextList_ConfigErrorAlarmTextLibrary_1": 1 'NameService configuration error: Implicit deletion. Subelement instance @6%s@ must be deleted explicitly.'; 2 'NameService configuration error: Implicit deletion. Alias/Format/Unit instance @6%s@ must be deleted explicitly.'

text list "SystemTextList_ConfigErrorAlarmTextLibrary_2": 1 'EvDpManager::cleanupDeletedDatapoint - alert handler config is deleted implicitly for deleted datapoint, @3%s@'; 2 'EvDpManager::cleanupDeletedDatapoint - alert handler config is deleted implicitly but still has overrides, @3%s@'; 3 'EvDpManager::cleanupDeletedDatapoint - default value config is deleted implicitly for deleted datapoint, @3%s@'; 4 'EvDpManager::cleanupDeletedDatapoint - default value config is deleted implicitly but still has overrides, @3%s@'; 5 'EvDpManager::cleanupDeletedDatapoint - initial value config is deleted implicitly for deleted datapoint, @3%s@'; 6 'EvDpManager::cleanupDeletedDatapoint - initial value config is deleted implicitly but still has overrides, @3%s@'; 7 'EvDpManager::cleanupDeletedDatapoint - distribution config is deleted implicitly for deleted datapoint, @3%s@'; 8 'EvDpManager::cleanupDeletedDatapoint - distribution config is deleted implicitly but still has overrides, @3%s@'; 9 'EvDpManager::cleanupDeletedDatapoint - rangeCheck config is deleted implicitly for deleted datapoint, @3%s@'; 10 'EvDpManager::cleanupDeletedDatapoint - rangeCheck config is deleted implicitly but still has overrides, @3%s@'

text list "SystemTextList_ConfigErrorAlarmTextLibrary_3": 1 'The configured data point type was deleted, but a configured type is still defined for the node type: @3%s@.'; 2 'The configured data point node type was deleted in the data point type, but a configured type is still defined for the element: @3%s@.'

text list "SystemTextList_ConfigErrorAlarmTextLibrary_4": 2 'Cycles: @6%s@ does not exist'; 3 'Alarms: @6%s@ exists already'; 4 'Tags: Address @6%s@ was rejected'; 1 'Connections: @6%s@ does not exist'; 5 'Tags: Acquisition mode @6%s@ is not supported.'; 6 'Cycles: @6%s@ was deleted but associated tags exist.'; 7 'Connections: @6%s@ was deleted but associated tags exist.'; 8 'Tags: Tag @6%s@ was rejected.'; 9 'Tags: Tag @6%s@ has an invalid value.'; 0 'Connections: Connection to @6%s@ could not be established.'; 65638 'Connections: Connection to @6%s@ could not be established.'; 65639 'Connections: @6%s@ disconnected.'; 65640 'Connections: Connection to the HMI device @6%s@ is lost.'; 65641 'Connections: Connection to the PLC @6%s@ is lost.'; 65541 'Connections: Timeout while establishing the connection to @6%s@.'; 65542 'Connections: @6%s@ faulty.'; 65543 'Connections: Connection to the HMI device disconnected. Connection @5%s@ was changed.'; 65544 'Connections: Connection to the HMI device disconnected. Driver property was changed for connection @5%s@.'

text list "SystemTextList_ConfigErrorAlarmTextLibrary_5": 1 'Connections: Lifecycle monitoring cycle must be shorter than the response time.'; 2 'Connections: Cyclic services are configured but not supported by the target device.'; 3 'Connections: Change-controlled reading is configured but not supported by the target device.'; 4 'Tags: The address @6%s@ does not exist in the PLC.'; 5 'Tags: The default conversion type for the address @6%s@ could not be determined.'; 6 'Tags: Invalid conversion type'; 7 'Cycles: Invalid conversion type. Conversion is not supported at HmiCycle.'; 4096 'Connections: Version of the address @6%s@ is not supported.'; 4097 'Connections: PROFIBUS address is not supported.'; 4098 'Connections: Softbus address is not supported.'; 4099 'Connections: Address type @6%s@ is not supported.'; 4100 'Connections: Invalid connection name @6%s@. Access point is being ignored.'; 4101 'Connections: Routing is not supported. @6%s@ is not used.'; 4102 'Connections: Routing is not supported. @6%s@ is not used.'; 4103 'Connections: Invalid IP address @6%s@'; 4104 'Connections: Invalid Named Connection @6%s@. Valid format: >VMD</>connection<'; 4105 'Connections: Invalid Named Connection @6%s@. VMD connection name is too long. Only 24 characters are permitted.'; 4106 'Connections: Invalid Named Connection @6%s@. Connection name is too long. Only 32 characters are permitted.'; 4107 'Connections: Rack number @6%s@ is outside of the permitted range (0..7)'; 4108 'Connections: Invalid Named Connection @6%s@. Rack is ignored.'; 4109 'Connections: Slot number @6%s@ is outside of the permitted range (0..31)'; 4110 'Connections: Invalid Named Connection @6%s@. Slot is ignored.'; 4111 'Connection could not be established. Maximum number of available connections (@6%s@) has been exceeded.'; 4112 'Connection aborted. No sign of life in the last @4%s@ ms.'; 4113 'Connection could not be established - @4%s@'; 4114 'Connection could not be established. The address @6%s@ cannot be used.'; 4115 'Connection could not be established. Invalid address @6%s@'; 4116 'Connection could not be established - @4%s@'

text list "SystemTextList_ConfigErrorAlarmTextLibrary_6": 1 'Connection could not be established. Application instance certificate is not configured.'; 2 'Connection could not be established. Server has rejected the client certificate. OPC UA status code @4%s@.'; 3 'Connection could not be established. Internal problem in the certificate store. OPC UA status code @4%s@'; 4 'Connection could not be established. Application instance certificate could not be loaded. OPC UA status code @4%s@'; 5 'Connection could not be established. Server has not provided a certificate. @4%s@'; 6 'Connection could not be established. Validation of server certificate has failed. OPC UA status code @4%s@.'; 7 'Connection was closed. Error during alarm synchronization. OPC UA status code @4%s@.'; 8 'Connection was closed. Alarm/event subscription has failed. The number of operations on the server has been exceeded.'; 9 'Connection was closed. Alarm/event subscription has failed. The number of alarm/event subscriptions on the server has been exceeded.'; 10 'Connection could not be established. Server reports a license problem. OPC UA status code @4%s@.'; 11 'Connection could not be established. Maximum number of server sessions has been exceeded.'; 12 'Connection could not be established. Safety configuration is inconsistent. @4%s@'; 13 'Connection could not be established. The address @4%s@ cannot be used.'; 14 'Connection could not be established. OPC UA status code @4%s@'; 15 'Connection aborted. OPC UA server was stopped.'; 16 'Connection aborted. No sign of life in the last @4%s@ ms.'; 17 'Connection was closed. OPC UA server maintenance.'; 18 'Connection could not be established. Invalid configuration of the authentication mode - @4%s@'; 19 'Connection could not be established. User could not be authenticated. OPC UA status code @4%s@'; 20 'Connection could not be established. Server does not permit anonymous connection. OPC UA status code @4%s@'; 21 'Connection could not be established. Certificate problem: Error when writing the safety-relevant data to @4%s@.'; 22 'Connection could not be established. Certificate problem: Unexpected file in the folder @4%s@ cannot be removed.'; 23 'Connection could not be established. User could not be authenticated. No user or password configured.'; 24 'Connection could not be established. Unexpected length of the server certificate. @4%s@'; 25 'Connection could not be established. @4%s@ is empty.'; 26 'Connection could not be established. @4%s@ has an unexpected format.'; 27 'Connection could not be established. Server endpoints cannot be read. OPC UA status code @4%s@'; 28 'Connection could not be established. No server endpoints were found. @4%s@'; 29 'Connection could not be established. Application instance certificate could not be found.'; 30 'Connection could not be established. Unexpected format of the certificate @4%s@.'; 31 'Connection could not be established. Unexpected format of the certificate block list @4%s@.'; 32 'Connection could not be established. User could not be authenticated. An encryption detail is invalid. @4%s@'; 34 'Connection could not be established. - The configured non-transparent redundancy mode @4%s@ is not supported.'; 101 'Tags: Address @6%s@ does not exist on the server.'; 103 'Tags: Address @6%s@ cannot be accessed.'; 104 'Tags: Acquisition mode is not supported for address @6%s@.'; 201 'Alarms: Address @6%s@ does not exist on the server.'; 202 'Alarms: Address @6%s@ cannot be used. The specified range filter is not an OPC UA Event Notifier.'; 203 'Alarms: Address @6%s@ cannot be used. The specified range filter does not exist on the server.'; 204 'Alarms: Address @6%s@ cannot be used because it is not an OPC UA event type.'; 205 'Alarms: Address @6%s@ cannot be used because the OPC UA condition type is not supported.'; 206 'Alarms: Address @6%s@ cannot be used because the event type does not exist on the server.'; 207 'Alarms: Acquisition type cannot be used for address @6%s@.'; 301 'Address @6%s@ cannot be used because the version number is missing.'; 302 'Address @6%s@ cannot be used because the version number is invalid.'; 303 'Address @6%s@ cannot be used because the number of '$' delimiters is invalid.'; 304 'Address @6%s@ cannot be used because the address type is invalid.'; 305 'Unsupported version @6%s@ of the address'; 401 'Unexpected OPC UA server response: @6%s@'

text list "SystemTextList_ConfigErrorAlarmTextLibrary_7": 1 'Messages: Invalid condition string for the alarm view @6%s@.'; 2 'Messages: Invalid status tag and bit for the alarm view @6%s@.'; 3 'Messages: Invalid control tag and bit for the alarm view @6%s@.'

text list "SystemTextList_ConfigErrorAlarmTextLibrary_8": 1 'Logs: Implicit deletion. Logging tag instance @6%s@ should be deleted but there are overloaded elements.'

text list "SystemTextList_ConfigErrorAlarmTextLibrary_9": 2 'Restart of the runtime is required.'; 3 'The correct storage medium must be ejected and inserted again.'

text list "SystemTextList_ConfigErrorAlarmTextLibrary_10": 1 'CDS cache - Cache folder cannot be created or reached: @6%s@'; 2 'LOC cache - Cache folder cannot be created or reached: @6%s@'

text list "SystemTextList_ConfigErrorAlarmTextLibrary_11": 2 'and synchronization will start automatically. Shutting down either of them during synchronization will not cause data loss.'; 3 'and synchronization is scheduled for: @5%Y-%m-%d %H:%M:%S@. Shutting down either of the computers will not cause data loss.'

text list "SystemTextList_RuntimeCollaborationFailureReason_1": 0 'Unknown error (@3%s@)'; 1 'The system is not running or there is a network problem'; 2 'Runtime is not started on the target device.'; 3 'The System ID does not match the expected System ID (@3%s@)'; 4 'The Collaboration name does not match the expected Collaboration name '@3%s@''; 5 'Wrong or unknown certificate'; 6 'Revoked certificate'; 7 'The time difference is too big.'; 8 'No common supported message version'; 9 'System ID (@3%s@) already exists'; 10 'System name (@3%s@) already exists'; 11 'ID/Name in local configuration for Runtime Collaboration already exists'

text list "SystemTextList_RedundancyRecoveryFailureReason_1": 0 'Data recovery request temporarily rejected until own recovery request has been responded to.'; 1 'Data recovery request rejected. Online backup running.'; 2 'Data recovery request rejected. Connection to the Event Manager is not established.'; 3 'Data recovery request temporarily rejected until delta activation is complete.'; 4 'Data recovery request temporarily rejected until alarms and tags are retentive.'; 5 'Data recovery request rejected. The obligatory file config.level.es is missing on the computer.'; 6 'Data recovery request was canceled by the Event Manager.'; 7 'The data synchronization between the devices has failed.'

text list "SystemTextList_S7PlusAlarmTextListCollection_1": 4096 'Connections: Connection to the PLC @4%s@ is lost'; 4097 'Connections: Connection to the HMI device @4%s@ is lost'; 4098 'Connections: Maximum number of connections exceeded - @4%s@'; 4099 'Out of resources on PLC - @4%s@'; 4100 'Legitimation failed, invalid or missing password - @4%s@'; 4101 'Request to open the connection failed - @4%s@'; 4102 'Connections: Cannot connect to PLC - @4%s@'; 4103 'Request to open the connection could not be sent'; 4104 'General certificate error for PLC - @4%s@'; 4105 'PLC certificate expired for PLC - @4%s@'; 4106 'PLC certificate is revoked for PLC - @4%s@'; 4107 'PLC certificate is untrustworthy. Manual trust is possible for - @4%s@'; 4108 'PLC certificate is untrustworthy. Manual trust is not possible for - @4%s@'

text list "SystemTextList_AllenBradleyEIPAlarmTextListCollection_7": 4096 'Connection lost on PLC side - @5%s@'; 4097 'Connection lost on HMI side - @5%s@'; 4098 'Maximum number of connections exceeded - @5%s@'; 4099 'Out of resources on PLC - @5%s@'; 4100 'Legitimation failed, invalid or missing password - @5%s@'; 4101 'Open request failed - @5%s@'; 4102 'Cannot connect to PLC - @5%s@'; 4103 'Open request could not be sent'; 4104 'root certificate expired for - @5%s@'; 4105 'PLC certificate untrusted for - @5%s@'

text list "SystemTextList_AllenBradleyDF1AlarmTextListCollection_9": 4096 'Connections: Connection to the PLC @5%s@ is lost'; 4097 'Connections: Connection to the HMI device @5%s@ is lost'; 4098 'Connections: Maximum number of connections exceeded - @5%s@'; 4099 'Out of resources on PLC - @5%s@'; 4100 'Legitimation failed, invalid or missing password - @5%s@'; 4101 'Request to open the connection failed - @5%s@'; 4102 'Connections: Cannot connect to PLC - @5%s@'; 4103 'Request to open the connection could not be sent'; 4104 'General certificate error for PLC - @5%s@'; 4105 'PLC certificate expired for PLC - @5%s@'; 4106 'PLC certificate is revoked for PLC - @5%s@'; 4107 'PLC certificate is untrustworthy. Manual trust is possible for - @5%s@'; 4108 'PLC certificate is untrustworthy. Manual trust is not possible for - @5%s@'

text list "SystemTextList_OmronEIPAlarmTextListCollection_6": 4096 'Connection lost on PLC side - @5%s@'; 4097 'Connection lost on HMI side - @5%s@'; 4098 'Maximum number of connections exceeded - @5%s@'; 4099 'Out of resources on PLC - @5%s@'; 4100 'Legitimation failed, invalid or missing password - @5%s@'; 4101 'Open request failed - @5%s@'; 4102 'Cannot connect to PLC - @5%s@'; 4103 'Open request could not be sent'; 4104 'root certificate expired for - @5%s@'; 4105 'PLC certificate untrusted for - @5%s@'

text list "SystemTextList_StdModbusTCPAlarmTextListCollection_5": 4096 'Connections: Connection to the PLC @5%s@ is lost'; 4097 'Connections: Connection to the HMI device @5%s@ is lost'; 4098 'Connections: Maximum number of connections exceeded - @5%s@'; 4099 'Out of resources on PLC - @5%s@'; 4100 'Legitimation failed, invalid or missing password - @5%s@'; 4101 'Request to open the connection failed - @5%s@'; 4102 'Connections: Cannot connect to PLC - @5%s@'; 4103 'Request to open the connection could not be sent'; 4104 'General certificate error for PLC - @5%s@'; 4105 'PLC certificate expired for PLC - @5%s@'; 4106 'PLC certificate is revoked for PLC - @5%s@'; 4107 'PLC certificate is untrustworthy. Manual trust is possible for - @5%s@'; 4108 'PLC certificate is untrustworthy. Manual trust is not possible for - @5%s@'

text list "SystemTextList_MitsubishiMCAlarmTextListCollection_4": 4096 'Connection lost on PLC side - @5%s@'; 4097 'Connection lost on HMI side - @5%s@'; 4098 'Maximum number of connections exceeded - @5%s@'; 4099 'Out of resources on PLC - @5%s@'; 4100 'Legitimation failed, invalid or missing password - @5%s@'; 4101 'Open request failed - @5%s@'; 4102 'Cannot connect to PLC - @5%s@'; 4103 'Open request could not be sent'; 4104 'root certificate expired for - @5%s@'; 4105 'PLC certificate untrusted for - @5%s@'

text list "SystemTextList_MitsubishiiQAlarmTextListCollection_3": 4096 'Connection lost on PLC side - @5%s@'; 4097 'Connection lost on HMI side - @5%s@'; 4098 'Maximum number of connections exceeded - @5%s@'; 4099 'Out of resources on PLC - @5%s@'; 4100 'Legitimation failed, invalid or missing password - @5%s@'; 4101 'Open request failed - @5%s@'; 4102 'Cannot connect to PLC - @5%s@'; 4103 'Open request could not be sent'; 4104 'root certificate expired for - @5%s@'; 4105 'PLC certificate untrusted for - @5%s@'

text list "SystemTextList_StdModbusRTUAlarmTextListCollection_8": 4096 'Connections: Connection to the PLC @5%s@ is lost'; 4097 'Connections: Connection to the HMI device @5%s@ is lost'; 4098 'Connections: Maximum number of connections exceeded - @5%s@'; 4099 'Out of resources on PLC - @5%s@'; 4100 'Legitimation failed, invalid or missing password - @5%s@'; 4101 'Request to open the connection failed - @5%s@'; 4102 'Connections: Cannot connect to PLC - @5%s@'; 4103 'Request to open the connection could not be sent'; 4104 'General certificate error for PLC - @5%s@'; 4105 'PLC certificate expired for PLC - @5%s@'; 4106 'PLC certificate is revoked for PLC - @5%s@'; 4107 'PLC certificate is untrustworthy. Manual trust is possible for - @5%s@'; 4108 'PLC certificate is untrustworthy. Manual trust is not possible for - @5%s@'

text list "SystemTextList_LogoAlarmTextListCollection_10": 4096 'Connections: Connection to the PLC @5%s@ is lost'; 4097 'Connections: Connection to the HMI device @5%s@ is lost'; 4098 'Connections: Maximum number of connections exceeded - @5%s@'; 4099 'Out of resources on PLC - @5%s@'; 4100 'Legitimation failed, invalid or missing password - @5%s@'; 4101 'Request to open the connection failed - @5%s@'; 4102 'Connections: Cannot connect to PLC - @5%s@'; 4103 'Request to open the connection could not be sent'; 4104 'General certificate error for PLC - @5%s@'; 4105 'PLC certificate expired for PLC - @5%s@'; 4106 'PLC certificate is revoked for PLC - @5%s@'; 4107 'PLC certificate is untrustworthy. Manual trust is possible for - @5%s@'; 4108 'PLC certificate is untrustworthy. Manual trust is not possible for - @5%s@'

graphic list "Switch": 0 'rotary-switches-open'; 1 'rotary-switches-close'

graphic list "Light": 0 'light_green_off'; 1 'light_green_on'

graphic list "Agitator": 0 'agitator_1'; 1 'agitator_2'; 2 'agitator_3'; 3 'agitator_4'
*)

(* ===== HMI "HMI_RT_2" =====
connection "Connection_2": ETHERNET, ILRT_S7_1500_OMS

HMI tags "01.PumpControl"
   "Stop" : Bool AT %M0.1, T100ms
   "Lo" : Bool AT %M0.2, T100ms
   "Start" : Bool AT %M0.0, T100ms
   "Hi" : Bool AT %M0.3, T100ms
   "P_1" : Bool AT %M0.4, T100ms
   "P_2" : Bool AT %M0.5, T100ms
   "P_3" : Bool AT %M0.6, T100ms
   "L" : Int AT %MW4, T100ms

HMI tags "02.BatchControl"
   "StartBatch" : Bool AT %M10.0, T100ms
   "StopBatch" : Bool AT %M10.1, T100ms
   "High" : Bool AT %M10.2, T100ms
   "Low" : Bool AT %M10.3, T100ms
   "Mixer" : Bool AT %M10.4, T100ms
   "Pump_A" : Bool AT %M10.5, T100ms
   "Pump_B" : Bool AT %M10.6, T100ms
   "Pump_P" : Bool AT %M10.7, T100ms
   "S_1" : Bool AT %M12.4, T100ms
   "S_2" : Bool AT %M12.5, T100ms
   "S_3" : Bool AT %M12.6, T100ms
   "S_4" : Bool AT %M12.7, T100ms
   "S_5" : Bool AT %M13.0, T100ms
   "S_6" : Bool AT %M13.1, T100ms
   "BatchActive" : Bool AT %M13.2, T100ms
   "Va" : Real AT %MD14, T100ms
   "Vb" : Real AT %MD18, T100ms
   "Va_SP" : Real AT %MD22, T100ms
   "Vb_SP" : Real AT %MD26, T100ms
   "ProductCnt" : Int AT %MW30, T100ms
   "ProductCnt_SP" : Int AT %MW32, T100ms
   "Level" : Int AT %MW34, T100ms
   "MixerPosition" : Int AT %MW36, T1s

text list "SystemTextList_ConfigErrorAlarmTextLibrary_1": 1 'NameService configuration error: Implicit deletion. Subelement instance @6%s@ must be deleted explicitly.'; 2 'NameService configuration error: Implicit deletion. Alias/Format/Unit instance @6%s@ must be deleted explicitly.'

text list "SystemTextList_ConfigErrorAlarmTextLibrary_2": 1 'EvDpManager::cleanupDeletedDatapoint - alert handler config is deleted implicitly for deleted datapoint, @3%s@'; 2 'EvDpManager::cleanupDeletedDatapoint - alert handler config is deleted implicitly but still has overrides, @3%s@'; 3 'EvDpManager::cleanupDeletedDatapoint - default value config is deleted implicitly for deleted datapoint, @3%s@'; 4 'EvDpManager::cleanupDeletedDatapoint - default value config is deleted implicitly but still has overrides, @3%s@'; 5 'EvDpManager::cleanupDeletedDatapoint - initial value config is deleted implicitly for deleted datapoint, @3%s@'; 6 'EvDpManager::cleanupDeletedDatapoint - initial value config is deleted implicitly but still has overrides, @3%s@'; 7 'EvDpManager::cleanupDeletedDatapoint - distribution config is deleted implicitly for deleted datapoint, @3%s@'; 8 'EvDpManager::cleanupDeletedDatapoint - distribution config is deleted implicitly but still has overrides, @3%s@'; 9 'EvDpManager::cleanupDeletedDatapoint - rangeCheck config is deleted implicitly for deleted datapoint, @3%s@'; 10 'EvDpManager::cleanupDeletedDatapoint - rangeCheck config is deleted implicitly but still has overrides, @3%s@'

text list "SystemTextList_ConfigErrorAlarmTextLibrary_3": 1 'The configured data point type was deleted, but a configured type is still defined for the node type: @3%s@.'; 2 'The configured data point node type was deleted in the data point type, but a configured type is still defined for the element: @3%s@.'

text list "SystemTextList_ConfigErrorAlarmTextLibrary_4": 2 'Cycles: @6%s@ does not exist'; 3 'Alarms: @6%s@ exists already'; 4 'Tags: Address @6%s@ was rejected'; 1 'Connections: @6%s@ does not exist'; 5 'Tags: Acquisition mode @6%s@ is not supported.'; 6 'Cycles: @6%s@ was deleted but associated tags exist.'; 7 'Connections: @6%s@ was deleted but associated tags exist.'; 8 'Tags: Tag @6%s@ was rejected.'; 9 'Tags: Tag @6%s@ has an invalid value.'; 0 'Connections: Connection to @6%s@ could not be established.'; 65638 'Connections: Connection to @6%s@ could not be established.'; 65639 'Connections: @6%s@ disconnected.'; 65640 'Connections: Connection to the HMI device @6%s@ is lost.'; 65641 'Connections: Connection to the PLC @6%s@ is lost.'; 65541 'Connections: Timeout while establishing the connection to @6%s@.'; 65542 'Connections: @6%s@ faulty.'; 65543 'Connections: Connection to the HMI device disconnected. Connection @5%s@ was changed.'; 65544 'Connections: Connection to the HMI device disconnected. Driver property was changed for connection @5%s@.'

text list "SystemTextList_ConfigErrorAlarmTextLibrary_5": 1 'Connections: Lifecycle monitoring cycle must be shorter than the response time.'; 2 'Connections: Cyclic services are configured but not supported by the target device.'; 3 'Connections: Change-controlled reading is configured but not supported by the target device.'; 4 'Tags: The address @6%s@ does not exist in the PLC.'; 5 'Tags: The default conversion type for the address @6%s@ could not be determined.'; 6 'Tags: Invalid conversion type'; 7 'Cycles: Invalid conversion type. Conversion is not supported at HmiCycle.'; 4096 'Connections: Version of the address @6%s@ is not supported.'; 4097 'Connections: PROFIBUS address is not supported.'; 4098 'Connections: Softbus address is not supported.'; 4099 'Connections: Address type @6%s@ is not supported.'; 4100 'Connections: Invalid connection name @6%s@. Access point is being ignored.'; 4101 'Connections: Routing is not supported. @6%s@ is not used.'; 4102 'Connections: Routing is not supported. @6%s@ is not used.'; 4103 'Connections: Invalid IP address @6%s@'; 4104 'Connections: Invalid Named Connection @6%s@. Valid format: >VMD</>connection<'; 4105 'Connections: Invalid Named Connection @6%s@. VMD connection name is too long. Only 24 characters are permitted.'; 4106 'Connections: Invalid Named Connection @6%s@. Connection name is too long. Only 32 characters are permitted.'; 4107 'Connections: Rack number @6%s@ is outside of the permitted range (0..7)'; 4108 'Connections: Invalid Named Connection @6%s@. Rack is ignored.'; 4109 'Connections: Slot number @6%s@ is outside of the permitted range (0..31)'; 4110 'Connections: Invalid Named Connection @6%s@. Slot is ignored.'; 4111 'Connection could not be established. Maximum number of available connections (@6%s@) has been exceeded.'; 4112 'Connection aborted. No sign of life in the last @4%s@ ms.'; 4113 'Connection could not be established - @4%s@'; 4114 'Connection could not be established. The address @6%s@ cannot be used.'; 4115 'Connection could not be established. Invalid address @6%s@'; 4116 'Connection could not be established - @4%s@'

text list "SystemTextList_ConfigErrorAlarmTextLibrary_6": 1 'Connection could not be established. Application instance certificate is not configured.'; 2 'Connection could not be established. Server has rejected the client certificate. OPC UA status code @4%s@.'; 3 'Connection could not be established. Internal problem in the certificate store. OPC UA status code @4%s@'; 4 'Connection could not be established. Application instance certificate could not be loaded. OPC UA status code @4%s@'; 5 'Connection could not be established. Server has not provided a certificate. @4%s@'; 6 'Connection could not be established. Validation of server certificate has failed. OPC UA status code @4%s@.'; 7 'Connection was closed. Error during alarm synchronization. OPC UA status code @4%s@.'; 8 'Connection was closed. Alarm/event subscription has failed. The number of operations on the server has been exceeded.'; 9 'Connection was closed. Alarm/event subscription has failed. The number of alarm/event subscriptions on the server has been exceeded.'; 10 'Connection could not be established. Server reports a license problem. OPC UA status code @4%s@.'; 11 'Connection could not be established. Maximum number of server sessions has been exceeded.'; 12 'Connection could not be established. Safety configuration is inconsistent. @4%s@'; 13 'Connection could not be established. The address @4%s@ cannot be used.'; 14 'Connection could not be established. OPC UA status code @4%s@'; 15 'Connection aborted. OPC UA server was stopped.'; 16 'Connection aborted. No sign of life in the last @4%s@ ms.'; 17 'Connection was closed. OPC UA server maintenance.'; 18 'Connection could not be established. Invalid configuration of the authentication mode - @4%s@'; 19 'Connection could not be established. User could not be authenticated. OPC UA status code @4%s@'; 20 'Connection could not be established. Server does not permit anonymous connection. OPC UA status code @4%s@'; 21 'Connection could not be established. Certificate problem: Error when writing the safety-relevant data to @4%s@.'; 22 'Connection could not be established. Certificate problem: Unexpected file in the folder @4%s@ cannot be removed.'; 23 'Connection could not be established. User could not be authenticated. No user or password configured.'; 24 'Connection could not be established. Unexpected length of the server certificate. @4%s@'; 25 'Connection could not be established. @4%s@ is empty.'; 26 'Connection could not be established. @4%s@ has an unexpected format.'; 27 'Connection could not be established. Server endpoints cannot be read. OPC UA status code @4%s@'; 28 'Connection could not be established. No server endpoints were found. @4%s@'; 29 'Connection could not be established. Application instance certificate could not be found.'; 30 'Connection could not be established. Unexpected format of the certificate @4%s@.'; 31 'Connection could not be established. Unexpected format of the certificate block list @4%s@.'; 32 'Connection could not be established. User could not be authenticated. An encryption detail is invalid. @4%s@'; 34 'Connection could not be established. - The configured non-transparent redundancy mode @4%s@ is not supported.'; 101 'Tags: Address @6%s@ does not exist on the server.'; 103 'Tags: Address @6%s@ cannot be accessed.'; 104 'Tags: Acquisition mode is not supported for address @6%s@.'; 201 'Alarms: Address @6%s@ does not exist on the server.'; 202 'Alarms: Address @6%s@ cannot be used. The specified range filter is not an OPC UA Event Notifier.'; 203 'Alarms: Address @6%s@ cannot be used. The specified range filter does not exist on the server.'; 204 'Alarms: Address @6%s@ cannot be used because it is not an OPC UA event type.'; 205 'Alarms: Address @6%s@ cannot be used because the OPC UA condition type is not supported.'; 206 'Alarms: Address @6%s@ cannot be used because the event type does not exist on the server.'; 207 'Alarms: Acquisition type cannot be used for address @6%s@.'; 301 'Address @6%s@ cannot be used because the version number is missing.'; 302 'Address @6%s@ cannot be used because the version number is invalid.'; 303 'Address @6%s@ cannot be used because the number of '$' delimiters is invalid.'; 304 'Address @6%s@ cannot be used because the address type is invalid.'; 305 'Unsupported version @6%s@ of the address'; 401 'Unexpected OPC UA server response: @6%s@'

text list "SystemTextList_ConfigErrorAlarmTextLibrary_7": 1 'Messages: Invalid condition string for the alarm view @6%s@.'; 2 'Messages: Invalid status tag and bit for the alarm view @6%s@.'; 3 'Messages: Invalid control tag and bit for the alarm view @6%s@.'

text list "SystemTextList_ConfigErrorAlarmTextLibrary_8": 1 'Logs: Implicit deletion. Logging tag instance @6%s@ should be deleted but there are overloaded elements.'

text list "SystemTextList_ConfigErrorAlarmTextLibrary_9": 2 'Restart of the runtime is required.'; 3 'The correct storage medium must be ejected and inserted again.'

text list "SystemTextList_ConfigErrorAlarmTextLibrary_10": 1 'CDS cache - Cache folder cannot be created or reached: @6%s@'; 2 'LOC cache - Cache folder cannot be created or reached: @6%s@'

text list "SystemTextList_ConfigErrorAlarmTextLibrary_11": 2 'and synchronization will start automatically. Shutting down either of them during synchronization will not cause data loss.'; 3 'and synchronization is scheduled for: @5%Y-%m-%d %H:%M:%S@. Shutting down either of the computers will not cause data loss.'

text list "SystemTextList_RuntimeCollaborationFailureReason_1": 0 'Unknown error (@3%s@)'; 1 'The system is not running or there is a network problem'; 2 'Runtime is not started on the target device.'; 3 'The System ID does not match the expected System ID (@3%s@)'; 4 'The Collaboration name does not match the expected Collaboration name '@3%s@''; 5 'Wrong or unknown certificate'; 6 'Revoked certificate'; 7 'The time difference is too big.'; 8 'No common supported message version'; 9 'System ID (@3%s@) already exists'; 10 'System name (@3%s@) already exists'; 11 'ID/Name in local configuration for Runtime Collaboration already exists'

text list "SystemTextList_RedundancyRecoveryFailureReason_1": 0 'Data recovery request temporarily rejected until own recovery request has been responded to.'; 1 'Data recovery request rejected. Online backup running.'; 2 'Data recovery request rejected. Connection to the Event Manager is not established.'; 3 'Data recovery request temporarily rejected until delta activation is complete.'; 4 'Data recovery request temporarily rejected until alarms and tags are retentive.'; 5 'Data recovery request rejected. The obligatory file config.level.es is missing on the computer.'; 6 'Data recovery request was canceled by the Event Manager.'; 7 'The data synchronization between the devices has failed.'

text list "SystemTextList_S7PlusAlarmTextListCollection_1": 4096 'Connections: Connection to the PLC @4%s@ is lost'; 4097 'Connections: Connection to the HMI device @4%s@ is lost'; 4098 'Connections: Maximum number of connections exceeded - @4%s@'; 4099 'Out of resources on PLC - @4%s@'; 4100 'Legitimation failed, invalid or missing password - @4%s@'; 4101 'Request to open the connection failed - @4%s@'; 4102 'Connections: Cannot connect to PLC - @4%s@'; 4103 'Request to open the connection could not be sent'; 4104 'General certificate error for PLC - @4%s@'; 4105 'PLC certificate expired for PLC - @4%s@'; 4106 'PLC certificate is revoked for PLC - @4%s@'; 4107 'PLC certificate is untrustworthy. Manual trust is possible for - @4%s@'; 4108 'PLC certificate is untrustworthy. Manual trust is not possible for - @4%s@'

text list "SystemTextList_AllenBradleyEIPAlarmTextListCollection_7": 4096 'Connection lost on PLC side - @5%s@'; 4097 'Connection lost on HMI side - @5%s@'; 4098 'Maximum number of connections exceeded - @5%s@'; 4099 'Out of resources on PLC - @5%s@'; 4100 'Legitimation failed, invalid or missing password - @5%s@'; 4101 'Open request failed - @5%s@'; 4102 'Cannot connect to PLC - @5%s@'; 4103 'Open request could not be sent'; 4104 'root certificate expired for - @5%s@'; 4105 'PLC certificate untrusted for - @5%s@'

text list "SystemTextList_AllenBradleyDF1AlarmTextListCollection_9": 4096 'Connections: Connection to the PLC @5%s@ is lost'; 4097 'Connections: Connection to the HMI device @5%s@ is lost'; 4098 'Connections: Maximum number of connections exceeded - @5%s@'; 4099 'Out of resources on PLC - @5%s@'; 4100 'Legitimation failed, invalid or missing password - @5%s@'; 4101 'Request to open the connection failed - @5%s@'; 4102 'Connections: Cannot connect to PLC - @5%s@'; 4103 'Request to open the connection could not be sent'; 4104 'General certificate error for PLC - @5%s@'; 4105 'PLC certificate expired for PLC - @5%s@'; 4106 'PLC certificate is revoked for PLC - @5%s@'; 4107 'PLC certificate is untrustworthy. Manual trust is possible for - @5%s@'; 4108 'PLC certificate is untrustworthy. Manual trust is not possible for - @5%s@'

text list "SystemTextList_OmronEIPAlarmTextListCollection_6": 4096 'Connection lost on PLC side - @5%s@'; 4097 'Connection lost on HMI side - @5%s@'; 4098 'Maximum number of connections exceeded - @5%s@'; 4099 'Out of resources on PLC - @5%s@'; 4100 'Legitimation failed, invalid or missing password - @5%s@'; 4101 'Open request failed - @5%s@'; 4102 'Cannot connect to PLC - @5%s@'; 4103 'Open request could not be sent'; 4104 'root certificate expired for - @5%s@'; 4105 'PLC certificate untrusted for - @5%s@'

text list "SystemTextList_StdModbusTCPAlarmTextListCollection_5": 4096 'Connections: Connection to the PLC @5%s@ is lost'; 4097 'Connections: Connection to the HMI device @5%s@ is lost'; 4098 'Connections: Maximum number of connections exceeded - @5%s@'; 4099 'Out of resources on PLC - @5%s@'; 4100 'Legitimation failed, invalid or missing password - @5%s@'; 4101 'Request to open the connection failed - @5%s@'; 4102 'Connections: Cannot connect to PLC - @5%s@'; 4103 'Request to open the connection could not be sent'; 4104 'General certificate error for PLC - @5%s@'; 4105 'PLC certificate expired for PLC - @5%s@'; 4106 'PLC certificate is revoked for PLC - @5%s@'; 4107 'PLC certificate is untrustworthy. Manual trust is possible for - @5%s@'; 4108 'PLC certificate is untrustworthy. Manual trust is not possible for - @5%s@'

text list "SystemTextList_MitsubishiMCAlarmTextListCollection_4": 4096 'Connection lost on PLC side - @5%s@'; 4097 'Connection lost on HMI side - @5%s@'; 4098 'Maximum number of connections exceeded - @5%s@'; 4099 'Out of resources on PLC - @5%s@'; 4100 'Legitimation failed, invalid or missing password - @5%s@'; 4101 'Open request failed - @5%s@'; 4102 'Cannot connect to PLC - @5%s@'; 4103 'Open request could not be sent'; 4104 'root certificate expired for - @5%s@'; 4105 'PLC certificate untrusted for - @5%s@'

text list "SystemTextList_MitsubishiiQAlarmTextListCollection_3": 4096 'Connection lost on PLC side - @5%s@'; 4097 'Connection lost on HMI side - @5%s@'; 4098 'Maximum number of connections exceeded - @5%s@'; 4099 'Out of resources on PLC - @5%s@'; 4100 'Legitimation failed, invalid or missing password - @5%s@'; 4101 'Open request failed - @5%s@'; 4102 'Cannot connect to PLC - @5%s@'; 4103 'Open request could not be sent'; 4104 'root certificate expired for - @5%s@'; 4105 'PLC certificate untrusted for - @5%s@'

text list "SystemTextList_StdModbusRTUAlarmTextListCollection_8": 4096 'Connections: Connection to the PLC @5%s@ is lost'; 4097 'Connections: Connection to the HMI device @5%s@ is lost'; 4098 'Connections: Maximum number of connections exceeded - @5%s@'; 4099 'Out of resources on PLC - @5%s@'; 4100 'Legitimation failed, invalid or missing password - @5%s@'; 4101 'Request to open the connection failed - @5%s@'; 4102 'Connections: Cannot connect to PLC - @5%s@'; 4103 'Request to open the connection could not be sent'; 4104 'General certificate error for PLC - @5%s@'; 4105 'PLC certificate expired for PLC - @5%s@'; 4106 'PLC certificate is revoked for PLC - @5%s@'; 4107 'PLC certificate is untrustworthy. Manual trust is possible for - @5%s@'; 4108 'PLC certificate is untrustworthy. Manual trust is not possible for - @5%s@'

text list "SystemTextList_LogoAlarmTextListCollection_10": 4096 'Connections: Connection to the PLC @5%s@ is lost'; 4097 'Connections: Connection to the HMI device @5%s@ is lost'; 4098 'Connections: Maximum number of connections exceeded - @5%s@'; 4099 'Out of resources on PLC - @5%s@'; 4100 'Legitimation failed, invalid or missing password - @5%s@'; 4101 'Request to open the connection failed - @5%s@'; 4102 'Connections: Cannot connect to PLC - @5%s@'; 4103 'Request to open the connection could not be sent'; 4104 'General certificate error for PLC - @5%s@'; 4105 'PLC certificate expired for PLC - @5%s@'; 4106 'PLC certificate is revoked for PLC - @5%s@'; 4107 'PLC certificate is untrustworthy. Manual trust is possible for - @5%s@'; 4108 'PLC certificate is untrustworthy. Manual trust is not possible for - @5%s@'

graphic list "Switch": 0 'rotary-switches-open'; 1 'rotary-switches-close'

graphic list "Light": 0 'light_green_off'; 1 'light_green_on'

graphic list "Agitator": 0 'agitator_1'; 1 'agitator_2'; 2 'agitator_3'; 3 'agitator_4'
*)

(* ===== HMI "HMI_RT_3" =====
connection "OOP_Connection": ETHERNET, ILRT_S7_1500_OMS

HMI tags "01.Flate"
   "Motor_1_Start" : Bool AT %DB1.DBX0.0, T100ms
   "Motor_1_Stop" : Bool AT %DB1.DBX0.1, T100ms
   "Motor_1_Cmd" : Bool AT %DB1.DBX2.0, T100ms
   "Motor_2_Start" : Bool AT %DB2.DBX0.0, T100ms
   "Motor_2_Stop" : Bool AT %DB2.DBX0.1, T100ms
   "Motor_2_Cmd" : Bool AT %DB2.DBX2.0, T100ms
   "Motor_3_Start" : Bool AT %DB3.DBX0.0, T100ms
   "Motor_3_Stop" : Bool AT %DB3.DBX0.1, T100ms
   "Motor_3_Cmd" : Bool AT %DB3.DBX2.0, T100ms

HMI tags "02.UDT&Faceplate"
   "Motor_1" : f64981b7-23c1-4b9c-90a3-7c9aa74d9c52 AT %DB4.DBX0.0, T100ms
   "Motor_2" : f64981b7-23c1-4b9c-90a3-7c9aa74d9c52 AT %DB5.DBX0.0, T100ms
   "Motor_3" : f64981b7-23c1-4b9c-90a3-7c9aa74d9c52 AT %DB6.DBX0.0, T100ms

